// Mitsubishi GX Works2 project: KME Straw Machine   PLC: FX3U/FX3UC

PROGRAM MAIN
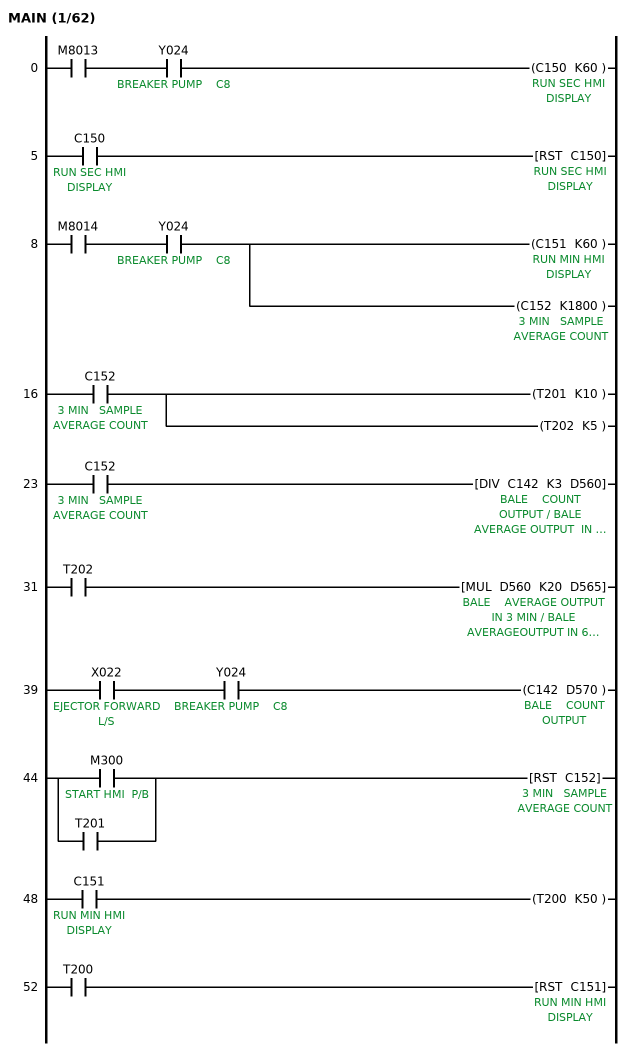
0     LD      M8013
      AND     Y024  ; BREAKER PUMP    C8
      OUT     C150 K60  ; RUN SEC HMI     DISPLAY
5     LD      C150  ; RUN SEC HMI     DISPLAY
      RST     C150  ; RUN SEC HMI     DISPLAY
8     LD      M8014
      AND     Y024  ; BREAKER PUMP    C8
      OUT     C151 K60  ; RUN MIN HMI     DISPLAY
      OUT     C152 K1800  ; 3 MIN   SAMPLE  AVERAGE COUNT
16    LD      C152  ; 3 MIN   SAMPLE  AVERAGE COUNT
      OUT     T201 K10
      OUT     T202 K5
23    LD      C152  ; 3 MIN   SAMPLE  AVERAGE COUNT
      DIV     C142 K3 D560  ; BALE    COUNT   OUTPUT / BALE    AVERAGE OUTPUT  IN 3 MIN
31    LD      T202
      MUL     D560 K20 D565  ; BALE     AVERAGEOUTPUT IN 60 MIN
39    LD      X022  ; EJECTOR FORWARD L/S
      AND     Y024  ; BREAKER PUMP    C8
      OUT     C142 D570  ; BALE    COUNT   OUTPUT
44    LD      M300  ; START HMI  P/B
      OR      T201
      RST     C152  ; 3 MIN   SAMPLE  AVERAGE COUNT
48    LD      C151  ; RUN MIN HMI     DISPLAY
      OUT     T200 K50
52    LD      T200
      RST     C151  ; RUN MIN HMI     DISPLAY
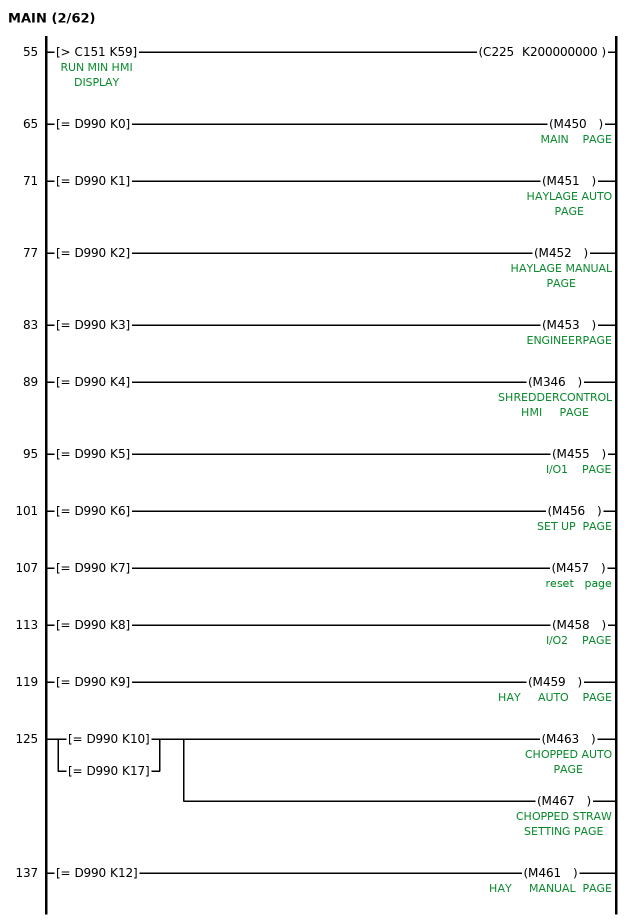
55    LD>     C151 K59  ; RUN MIN HMI     DISPLAY
      OUT     C225 K200000000
65    LD=     D990 K0
      OUT     M450  ; MAIN    PAGE
71    LD=     D990 K1
      OUT     M451  ; HAYLAGE AUTO    PAGE
77    LD=     D990 K2
      OUT     M452  ; HAYLAGE MANUAL  PAGE
83    LD=     D990 K3
      OUT     M453  ; ENGINEERPAGE
89    LD=     D990 K4
      OUT     M346  ; SHREDDERCONTROL HMI     PAGE
95    LD=     D990 K5
      OUT     M455  ; I/O1    PAGE
101   LD=     D990 K6
      OUT     M456  ; SET UP  PAGE
107   LD=     D990 K7
      OUT     M457  ; reset   page
113   LD=     D990 K8
      OUT     M458  ; I/O2    PAGE
119   LD=     D990 K9
      OUT     M459  ; HAY     AUTO    PAGE
125   LD=     D990 K10
      OR=     D990 K17
      OUT     M463  ; CHOPPED AUTO    PAGE
      OUT     M467  ; CHOPPED STRAW   SETTING PAGE
137   LD=     D990 K12
      OUT     M461  ; HAY     MANUAL  PAGE
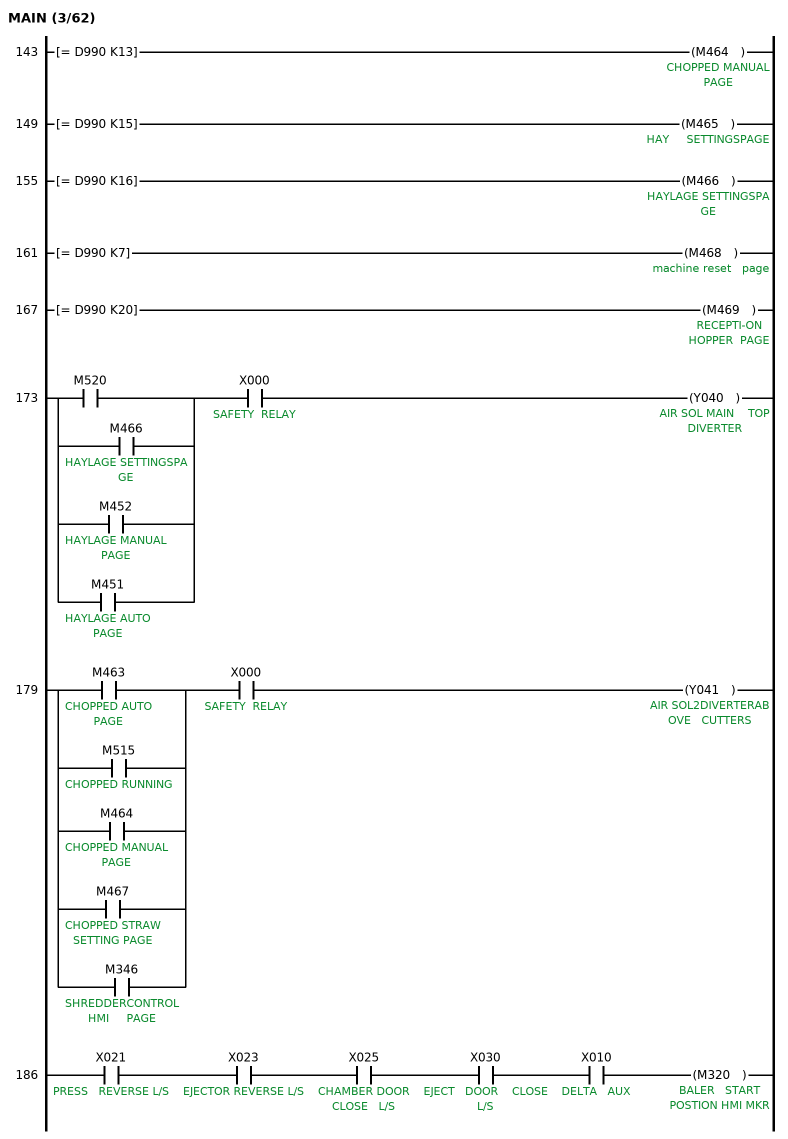
143   LD=     D990 K13
      OUT     M464  ; CHOPPED MANUAL  PAGE
149   LD=     D990 K15
      OUT     M465  ; HAY     SETTINGSPAGE
155   LD=     D990 K16
      OUT     M466  ; HAYLAGE SETTINGSPAGE
161   LD=     D990 K7
      OUT     M468  ; machine reset   page
167   LD=     D990 K20
      OUT     M469  ; RECEPTI-ON      HOPPER  PAGE
173   LD      M520
      OR      M466  ; HAYLAGE SETTINGSPAGE
      OR      M452  ; HAYLAGE MANUAL  PAGE
      OR      M451  ; HAYLAGE AUTO    PAGE
      AND     X000  ; SAFETY  RELAY
      OUT     Y040  ; AIR SOL MAIN    TOP     DIVERTER
179   LD      M463  ; CHOPPED AUTO    PAGE
      OR      M515  ; CHOPPED RUNNING
      OR      M464  ; CHOPPED MANUAL  PAGE
      OR      M467  ; CHOPPED STRAW   SETTING PAGE
      OR      M346  ; SHREDDERCONTROL HMI     PAGE
      AND     X000  ; SAFETY  RELAY
      OUT     Y041  ; AIR SOL2DIVERTERABOVE   CUTTERS
186   LD      X021  ; PRESS   REVERSE L/S
      AND     X023  ; EJECTOR REVERSE L/S
      AND     X025  ; CHAMBER DOOR    CLOSE   L/S
      AND     X030  ; EJECT   DOOR    CLOSE L/S
      AND     X010  ; DELTA   AUX
      OUT     M320  ; BALER   START   POSTION HMI MKR
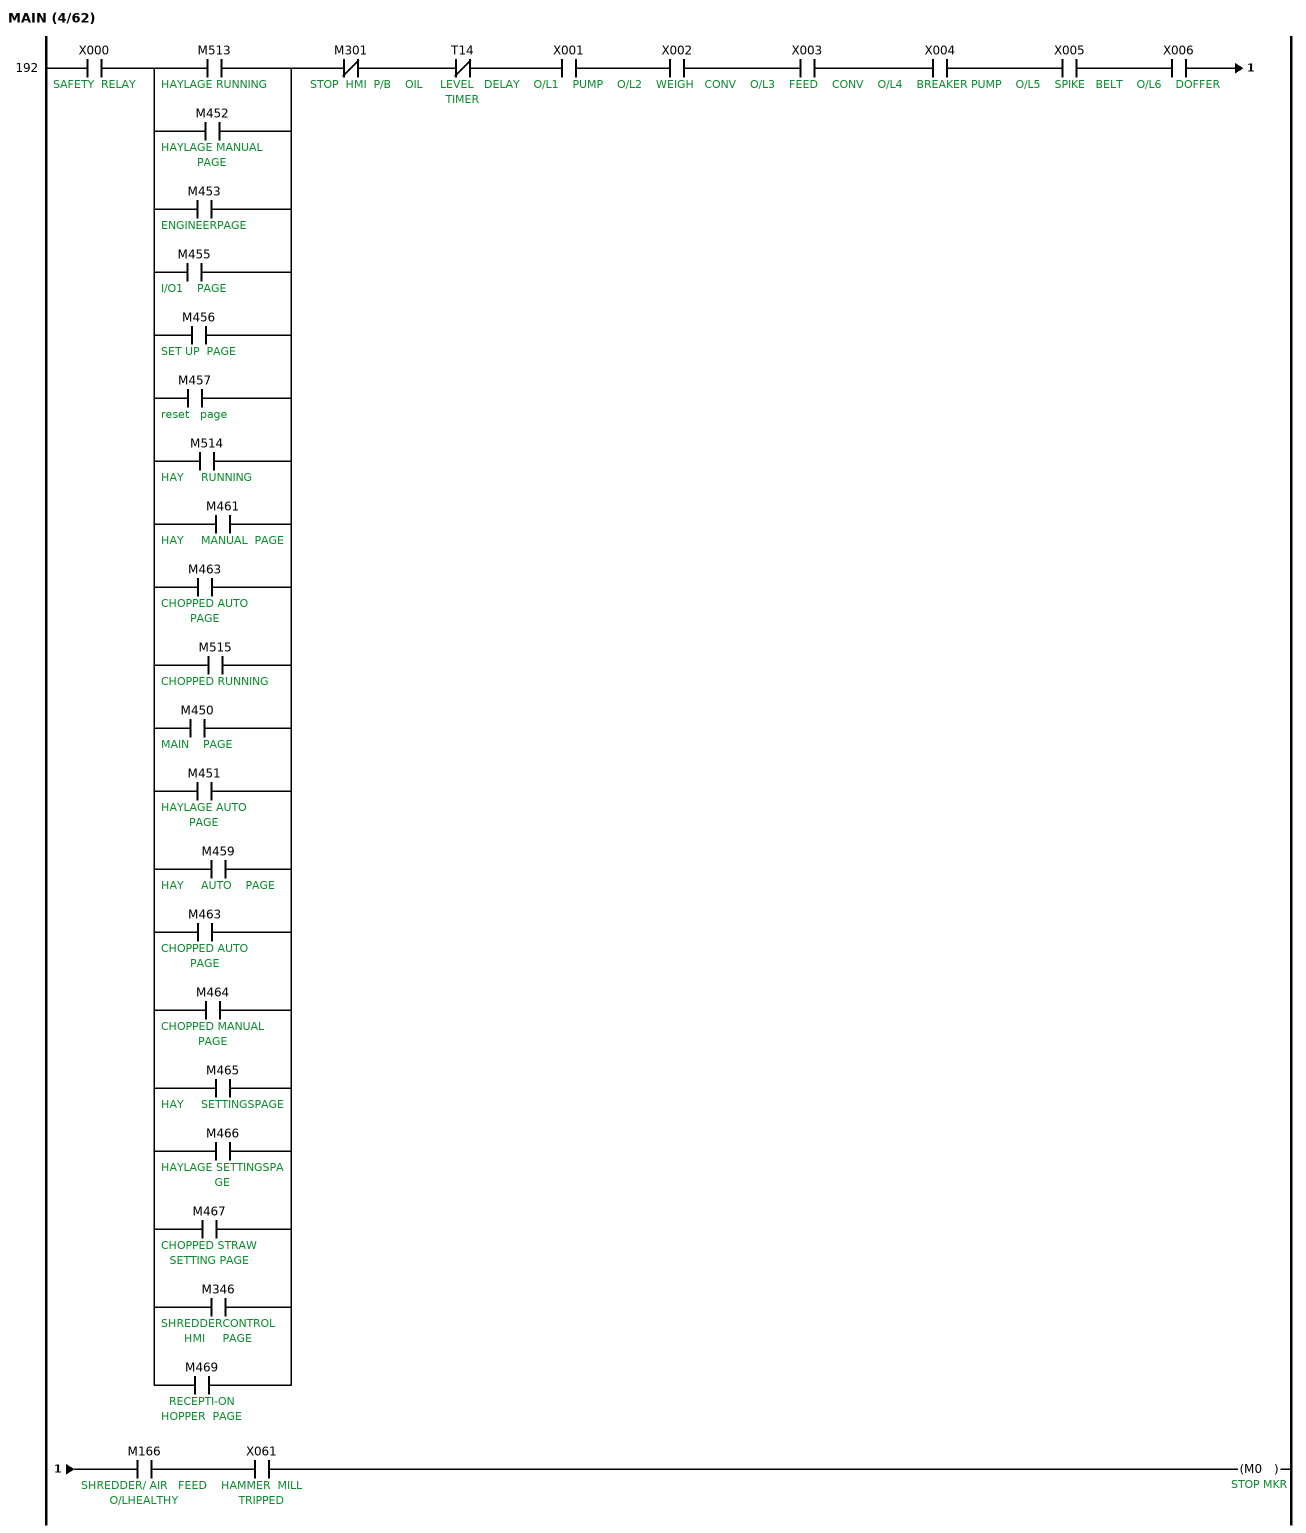
192   LD      X000  ; SAFETY  RELAY
      LD      M513  ; HAYLAGE RUNNING
      OR      M452  ; HAYLAGE MANUAL  PAGE
      OR      M453  ; ENGINEERPAGE
      OR      M455  ; I/O1    PAGE
      OR      M456  ; SET UP  PAGE
      OR      M457  ; reset   page
      OR      M514  ; HAY     RUNNING
      OR      M461  ; HAY     MANUAL  PAGE
      OR      M463  ; CHOPPED AUTO    PAGE
      OR      M515  ; CHOPPED RUNNING
      OR      M450  ; MAIN    PAGE
      OR      M451  ; HAYLAGE AUTO    PAGE
      OR      M459  ; HAY     AUTO    PAGE
      OR      M463  ; CHOPPED AUTO    PAGE
      OR      M464  ; CHOPPED MANUAL  PAGE
      OR      M465  ; HAY     SETTINGSPAGE
      OR      M466  ; HAYLAGE SETTINGSPAGE
      OR      M467  ; CHOPPED STRAW   SETTING PAGE
      OR      M346  ; SHREDDERCONTROL HMI     PAGE
      OR      M469  ; RECEPTI-ON      HOPPER  PAGE
      ANB
      ANI     M301  ; STOP  HMI  P/B
      ANI     T14  ; OIL     LEVEL   DELAY   TIMER
      AND     X001  ; O/L1    PUMP
      AND     X002  ; O/L2    WEIGH   CONV
      AND     X003  ; O/L3    FEED    CONV
      AND     X004  ; O/L4    BREAKER PUMP
      AND     X005  ; O/L5    SPIKE   BELT
      AND     X006  ; O/L6    DOFFER
      AND     M166  ; SHREDDER/ AIR   FEED O/LHEALTHY
      AND     X061  ; HAMMER  MILL    TRIPPED
      OUT     M0  ; STOP MKR
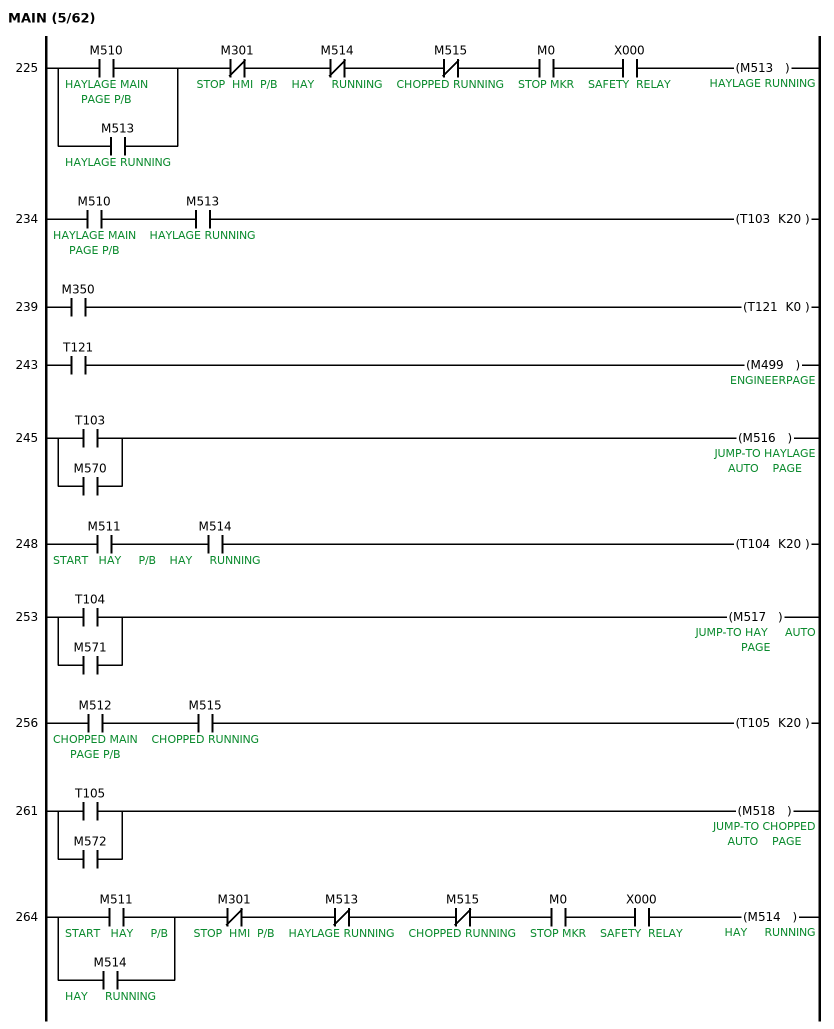
225   LD      M510  ; HAYLAGE MAIN    PAGE P/B
      OR      M513  ; HAYLAGE RUNNING
      ANI     M301  ; STOP  HMI  P/B
      ANI     M514  ; HAY     RUNNING
      ANI     M515  ; CHOPPED RUNNING
      AND     M0  ; STOP MKR
      AND     X000  ; SAFETY  RELAY
      OUT     M513  ; HAYLAGE RUNNING
234   LD      M510  ; HAYLAGE MAIN    PAGE P/B
      AND     M513  ; HAYLAGE RUNNING
      OUT     T103 K20
239   LD      M350
      OUT     T121 K0
243   LD      T121
      OUT     M499  ; ENGINEERPAGE
245   LD      T103
      OR      M570
      OUT     M516  ; JUMP-TO HAYLAGE AUTO    PAGE
248   LD      M511  ; START   HAY     P/B
      AND     M514  ; HAY     RUNNING
      OUT     T104 K20
253   LD      T104
      OR      M571
      OUT     M517  ; JUMP-TO HAY     AUTO    PAGE
256   LD      M512  ; CHOPPED MAIN    PAGE P/B
      AND     M515  ; CHOPPED RUNNING
      OUT     T105 K20
261   LD      T105
      OR      M572
      OUT     M518  ; JUMP-TO CHOPPED AUTO    PAGE
264   LD      M511  ; START   HAY     P/B
      OR      M514  ; HAY     RUNNING
      ANI     M301  ; STOP  HMI  P/B
      ANI     M513  ; HAYLAGE RUNNING
      ANI     M515  ; CHOPPED RUNNING
      AND     M0  ; STOP MKR
      AND     X000  ; SAFETY  RELAY
      OUT     M514  ; HAY     RUNNING
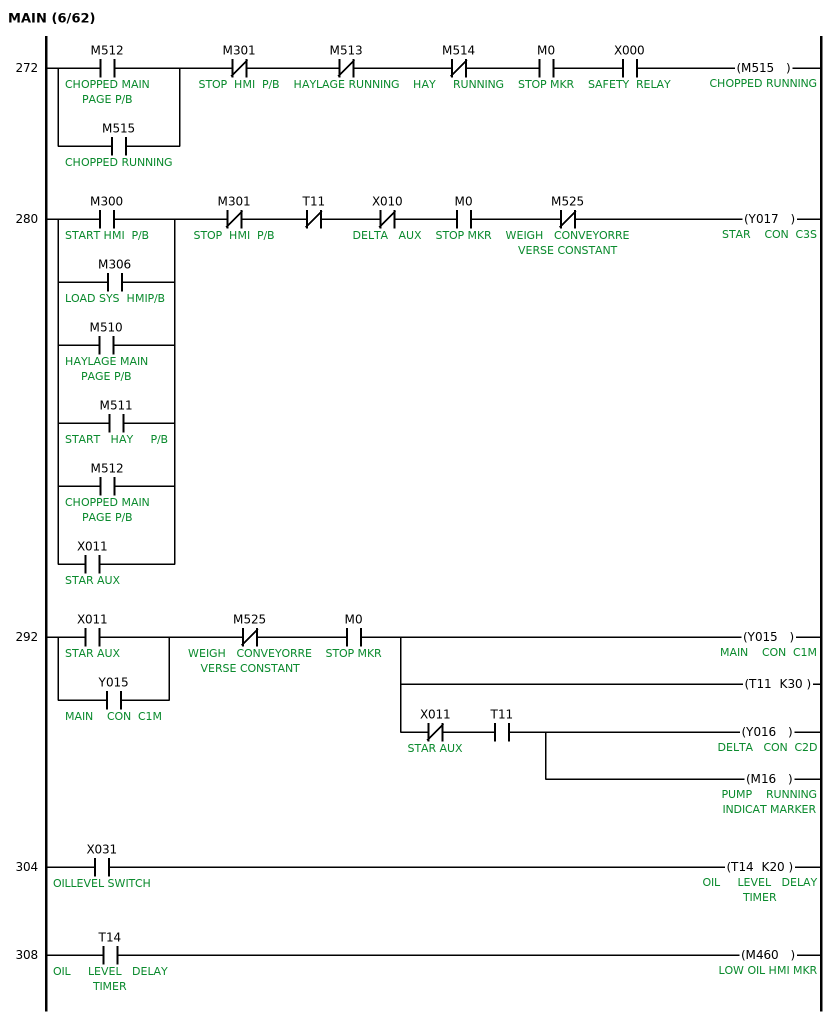
272   LD      M512  ; CHOPPED MAIN    PAGE P/B
      OR      M515  ; CHOPPED RUNNING
      ANI     M301  ; STOP  HMI  P/B
      ANI     M513  ; HAYLAGE RUNNING
      ANI     M514  ; HAY     RUNNING
      AND     M0  ; STOP MKR
      AND     X000  ; SAFETY  RELAY
      OUT     M515  ; CHOPPED RUNNING
280   LD      M300  ; START HMI  P/B
      OR      M306  ; LOAD SYS  HMIP/B
      OR      M510  ; HAYLAGE MAIN    PAGE P/B
      OR      M511  ; START   HAY     P/B
      OR      M512  ; CHOPPED MAIN    PAGE P/B
      OR      X011  ; STAR AUX
      ANI     M301  ; STOP  HMI  P/B
      ANI     T11
      ANI     X010  ; DELTA   AUX
      AND     M0  ; STOP MKR
      ANI     M525  ; WEIGH   CONVEYORREVERSE CONSTANT
      OUT     Y017  ; STAR    CON  C3S
292   LD      X011  ; STAR AUX
      OR      Y015  ; MAIN    CON  C1M
      ANI     M525  ; WEIGH   CONVEYORREVERSE CONSTANT
      AND     M0  ; STOP MKR
      OUT     Y015  ; MAIN    CON  C1M
      OUT     T11 K30
      ANI     X011  ; STAR AUX
      AND     T11
      OUT     Y016  ; DELTA   CON  C2D
      OUT     M16  ; PUMP    RUNNING INDICAT MARKER
304   LD      X031  ; OILLEVEL SWITCH
      OUT     T14 K20  ; OIL     LEVEL   DELAY   TIMER
308   LD      T14  ; OIL     LEVEL   DELAY   TIMER
      OUT     M460  ; LOW OIL HMI MKR
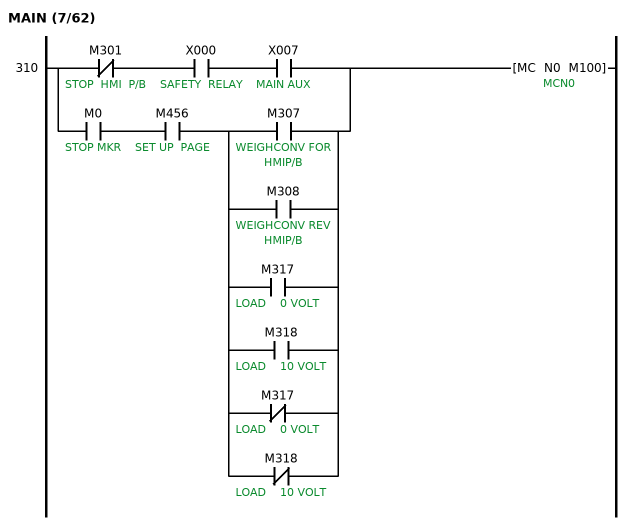
310   LDI     M301  ; STOP  HMI  P/B
      AND     X000  ; SAFETY  RELAY
      AND     X007  ; MAIN AUX
      LD      M0  ; STOP MKR
      AND     M456  ; SET UP  PAGE
      LD      M307  ; WEIGHCONV FOR   HMIP/B
      OR      M308  ; WEIGHCONV REV   HMIP/B
      OR      M317  ; LOAD    0 VOLT
      OR      M318  ; LOAD    10 VOLT
      ORI     M317  ; LOAD    0 VOLT
      ORI     M318  ; LOAD    10 VOLT
      ANB
      ORB
      MC      N0 M100  ; MCN0
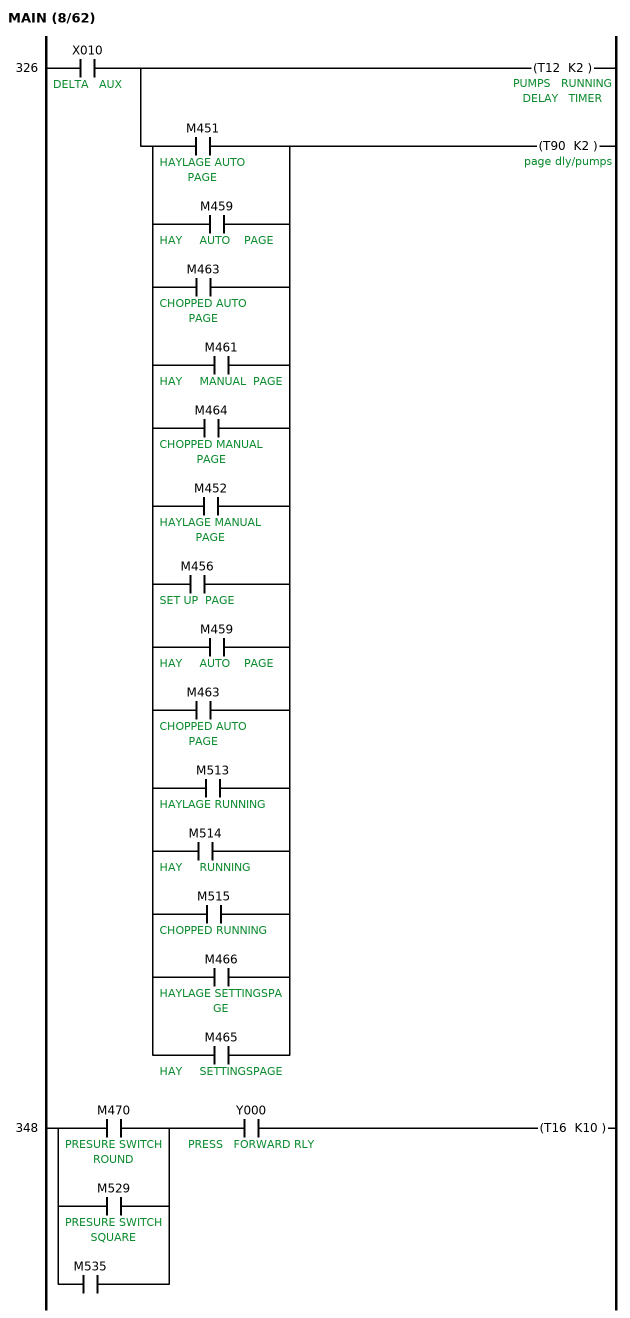
326   LD      X010  ; DELTA   AUX
      OUT     T12 K2  ; PUMPS   RUNNING DELAY   TIMER
      LD      M451  ; HAYLAGE AUTO    PAGE
      OR      M459  ; HAY     AUTO    PAGE
      OR      M463  ; CHOPPED AUTO    PAGE
      OR      M461  ; HAY     MANUAL  PAGE
      OR      M464  ; CHOPPED MANUAL  PAGE
      OR      M452  ; HAYLAGE MANUAL  PAGE
      OR      M456  ; SET UP  PAGE
      OR      M459  ; HAY     AUTO    PAGE
      OR      M463  ; CHOPPED AUTO    PAGE
      OR      M513  ; HAYLAGE RUNNING
      OR      M514  ; HAY     RUNNING
      OR      M515  ; CHOPPED RUNNING
      OR      M466  ; HAYLAGE SETTINGSPAGE
      OR      M465  ; HAY     SETTINGSPAGE
      ANB
      OUT     T90 K2  ; page dly/pumps
348   LD      M470  ; PRESURE SWITCH  ROUND
      OR      M529  ; PRESURE SWITCH  SQUARE
      OR      M535
      AND     Y000  ; PRESS   FORWARD RLY
      OUT     T16 K10
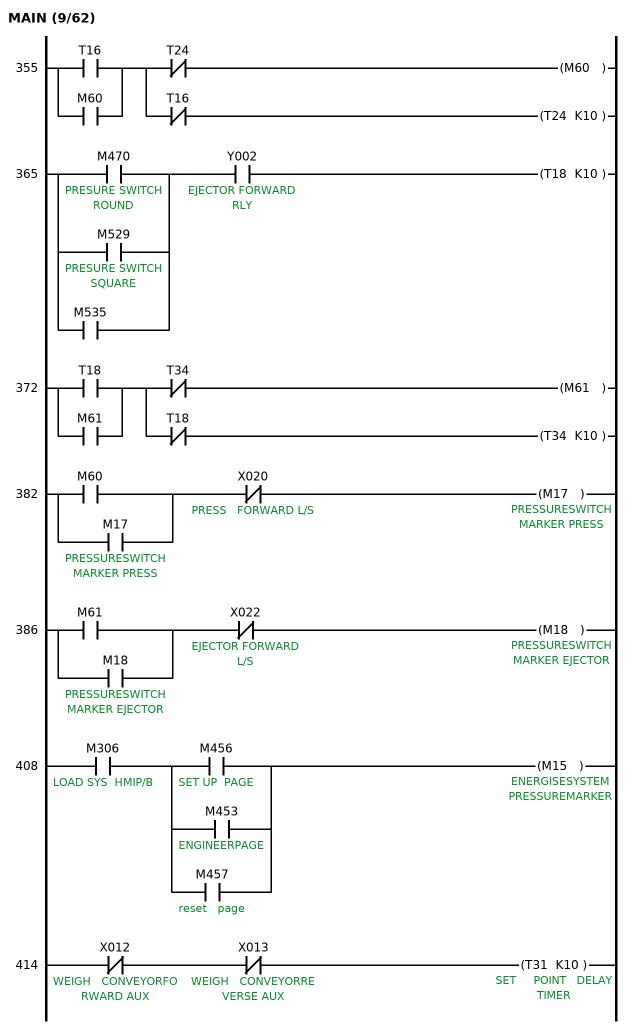
355   LD      T16
      OR      M60
      MPS
      ANI     T24
      OUT     M60
      MPP
      ANI     T16
      OUT     T24 K10
365   LD      M470  ; PRESURE SWITCH  ROUND
      OR      M529  ; PRESURE SWITCH  SQUARE
      OR      M535
      AND     Y002  ; EJECTOR FORWARD RLY
      OUT     T18 K10
372   LD      T18
      OR      M61
      MPS
      ANI     T34
      OUT     M61
      MPP
      ANI     T18
      OUT     T34 K10
382   LD      M60
      OR      M17  ; PRESSURESWITCH  MARKER PRESS
      ANI     X020  ; PRESS   FORWARD L/S
      OUT     M17  ; PRESSURESWITCH  MARKER PRESS
386   LD      M61
      OR      M18  ; PRESSURESWITCH  MARKER EJECTOR
      ANI     X022  ; EJECTOR FORWARD L/S
      OUT     M18  ; PRESSURESWITCH  MARKER EJECTOR
408   LD      M306  ; LOAD SYS  HMIP/B
      LD      M456  ; SET UP  PAGE
      OR      M453  ; ENGINEERPAGE
      OR      M457  ; reset   page
      ANB
      OUT     M15  ; ENERGISESYSTEM  PRESSUREMARKER
414   LDI     X012  ; WEIGH   CONVEYORFORWARD AUX
      ANI     X013  ; WEIGH   CONVEYORREVERSE AUX
      OUT     T31 K10  ; SET     POINT   DELAY   TIMER
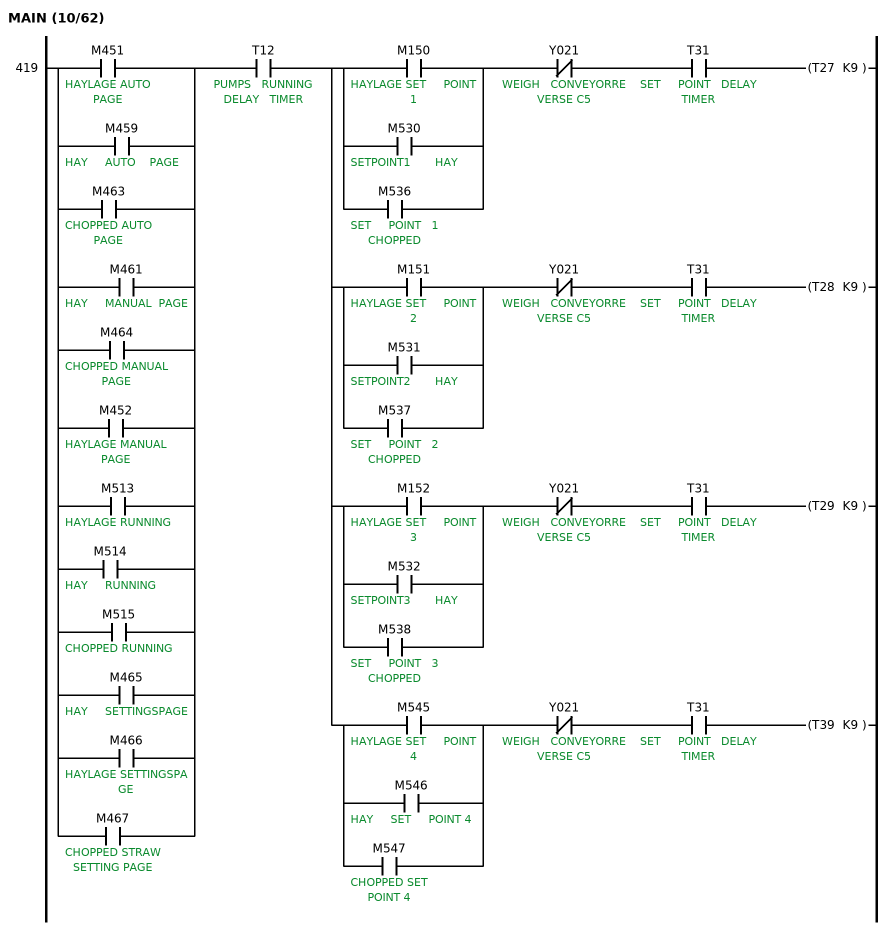
419   LD      M451  ; HAYLAGE AUTO    PAGE
      OR      M459  ; HAY     AUTO    PAGE
      OR      M463  ; CHOPPED AUTO    PAGE
      OR      M461  ; HAY     MANUAL  PAGE
      OR      M464  ; CHOPPED MANUAL  PAGE
      OR      M452  ; HAYLAGE MANUAL  PAGE
      OR      M513  ; HAYLAGE RUNNING
      OR      M514  ; HAY     RUNNING
      OR      M515  ; CHOPPED RUNNING
      OR      M465  ; HAY     SETTINGSPAGE
      OR      M466  ; HAYLAGE SETTINGSPAGE
      OR      M467  ; CHOPPED STRAW   SETTING PAGE
      AND     T12  ; PUMPS   RUNNING DELAY   TIMER
      MPS
      LD      M150  ; HAYLAGE SET     POINT 1
      OR      M530  ; SETPOINT1       HAY
      OR      M536  ; SET     POINT   1       CHOPPED
      ANB
      ANI     Y021  ; WEIGH   CONVEYORREVERSE C5
      AND     T31  ; SET     POINT   DELAY   TIMER
      OUT     T27 K9
      MRD
      LD      M151  ; HAYLAGE SET     POINT 2
      OR      M531  ; SETPOINT2       HAY
      OR      M537  ; SET     POINT   2       CHOPPED
      ANB
      ANI     Y021  ; WEIGH   CONVEYORREVERSE C5
      AND     T31  ; SET     POINT   DELAY   TIMER
      OUT     T28 K9
      MRD
      LD      M152  ; HAYLAGE SET     POINT 3
      OR      M532  ; SETPOINT3       HAY
      OR      M538  ; SET     POINT   3       CHOPPED
      ANB
      ANI     Y021  ; WEIGH   CONVEYORREVERSE C5
      AND     T31  ; SET     POINT   DELAY   TIMER
      OUT     T29 K9
      MPP
      LD      M545  ; HAYLAGE SET     POINT 4
      OR      M546  ; HAY     SET     POINT 4
      OR      M547  ; CHOPPED SET     POINT 4
      ANB
      ANI     Y021  ; WEIGH   CONVEYORREVERSE C5
      AND     T31  ; SET     POINT   DELAY   TIMER
      OUT     T39 K9
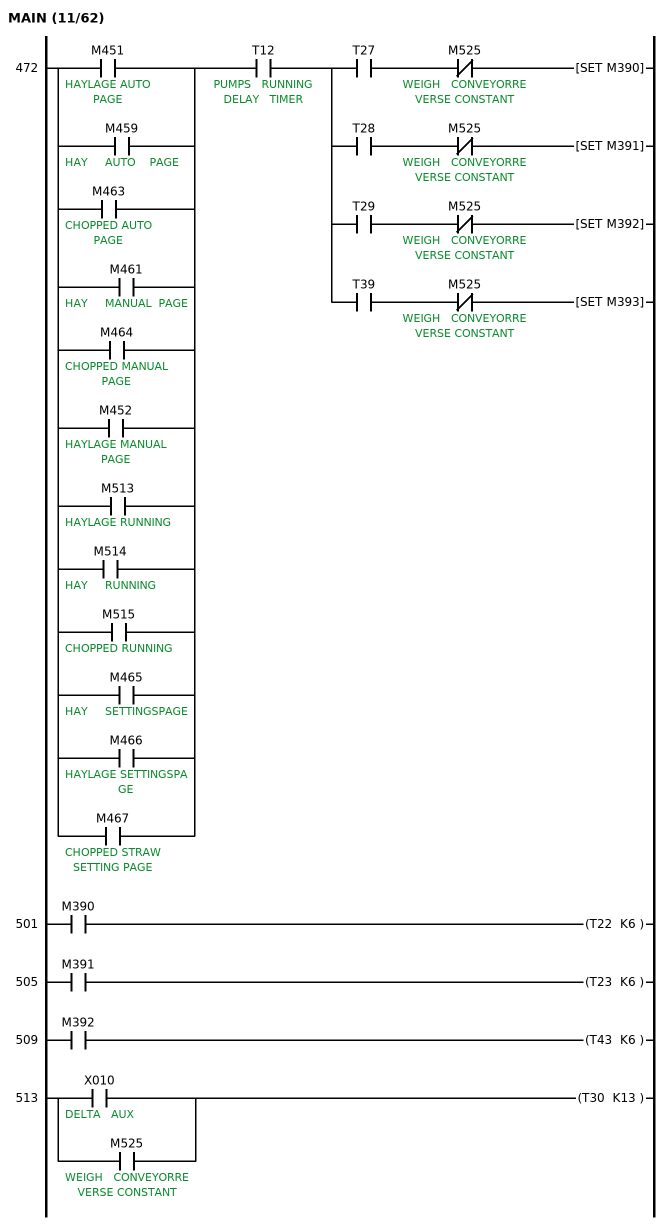
472   LD      M451  ; HAYLAGE AUTO    PAGE
      OR      M459  ; HAY     AUTO    PAGE
      OR      M463  ; CHOPPED AUTO    PAGE
      OR      M461  ; HAY     MANUAL  PAGE
      OR      M464  ; CHOPPED MANUAL  PAGE
      OR      M452  ; HAYLAGE MANUAL  PAGE
      OR      M513  ; HAYLAGE RUNNING
      OR      M514  ; HAY     RUNNING
      OR      M515  ; CHOPPED RUNNING
      OR      M465  ; HAY     SETTINGSPAGE
      OR      M466  ; HAYLAGE SETTINGSPAGE
      OR      M467  ; CHOPPED STRAW   SETTING PAGE
      AND     T12  ; PUMPS   RUNNING DELAY   TIMER
      MPS
      AND     T27
      ANI     M525  ; WEIGH   CONVEYORREVERSE CONSTANT
      SET     M390
      MRD
      AND     T28
      ANI     M525  ; WEIGH   CONVEYORREVERSE CONSTANT
      SET     M391
      MRD
      AND     T29
      ANI     M525  ; WEIGH   CONVEYORREVERSE CONSTANT
      SET     M392
      MPP
      AND     T39
      ANI     M525  ; WEIGH   CONVEYORREVERSE CONSTANT
      SET     M393
501   LD      M390
      OUT     T22 K6
505   LD      M391
      OUT     T23 K6
509   LD      M392
      OUT     T43 K6
513   LD      X010  ; DELTA   AUX
      OR      M525  ; WEIGH   CONVEYORREVERSE CONSTANT
      OUT     T30 K13
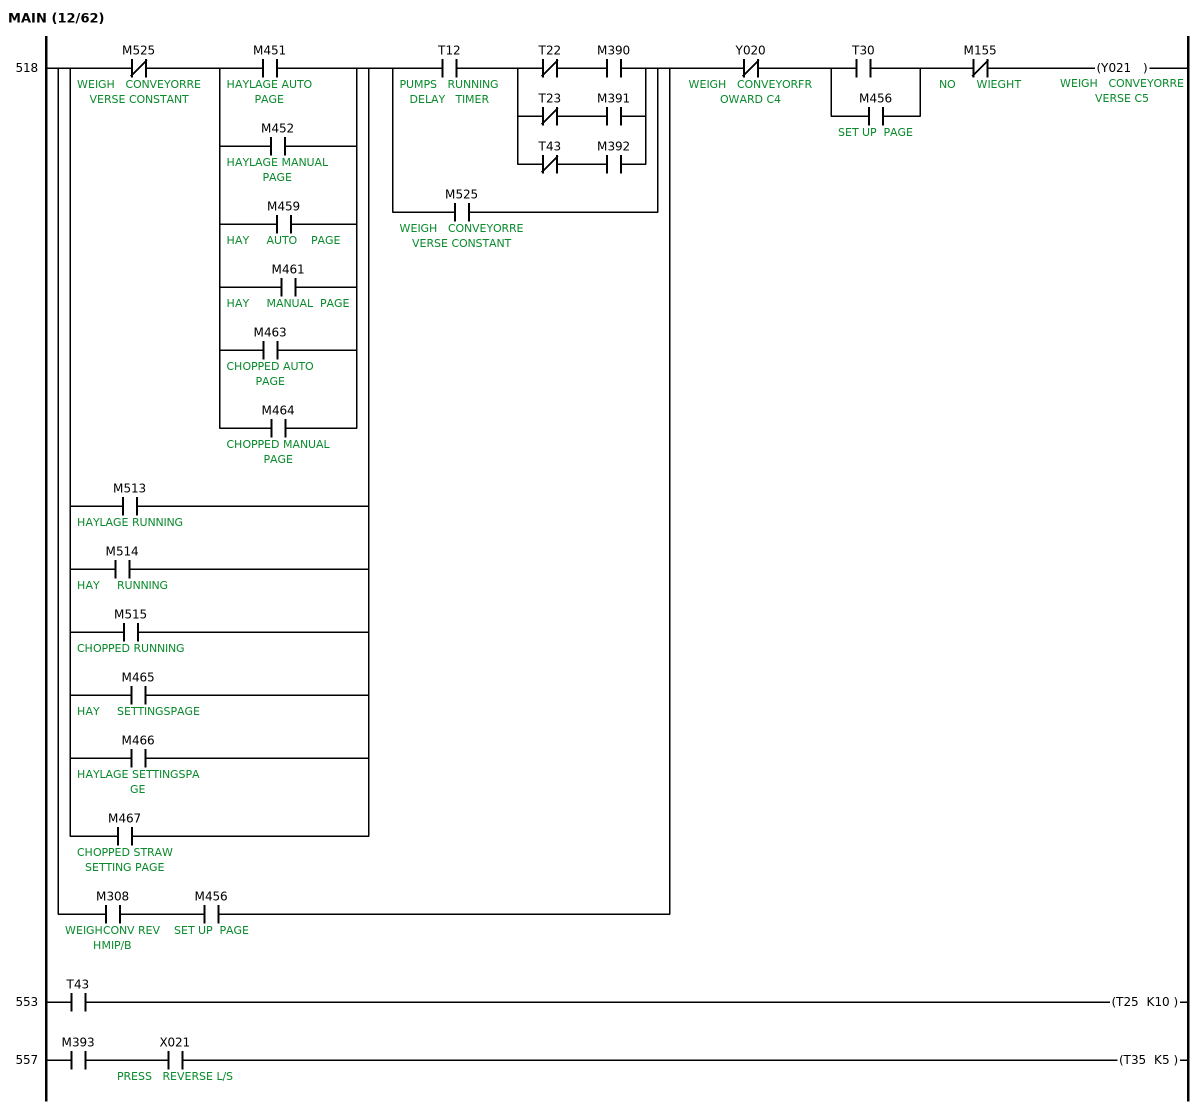
518   LDI     M525  ; WEIGH   CONVEYORREVERSE CONSTANT
      LD      M451  ; HAYLAGE AUTO    PAGE
      OR      M452  ; HAYLAGE MANUAL  PAGE
      OR      M459  ; HAY     AUTO    PAGE
      OR      M461  ; HAY     MANUAL  PAGE
      OR      M463  ; CHOPPED AUTO    PAGE
      OR      M464  ; CHOPPED MANUAL  PAGE
      ANB
      OR      M513  ; HAYLAGE RUNNING
      OR      M514  ; HAY     RUNNING
      OR      M515  ; CHOPPED RUNNING
      OR      M465  ; HAY     SETTINGSPAGE
      OR      M466  ; HAYLAGE SETTINGSPAGE
      OR      M467  ; CHOPPED STRAW   SETTING PAGE
      LD      T12  ; PUMPS   RUNNING DELAY   TIMER
      LDI     T22
      AND     M390
      LDI     T23
      AND     M391
      ORB
      LDI     T43
      AND     M392
      ORB
      ANB
      OR      M525  ; WEIGH   CONVEYORREVERSE CONSTANT
      ANB
      LD      M308  ; WEIGHCONV REV   HMIP/B
      AND     M456  ; SET UP  PAGE
      ORB
      ANI     Y020  ; WEIGH   CONVEYORFROWARD C4
      LD      T30
      OR      M456  ; SET UP  PAGE
      ANB
      ANI     M155  ; NO      WIEGHT
      OUT     Y021  ; WEIGH   CONVEYORREVERSE C5
553   LD      T43
      OUT     T25 K10
557   LD      M393
      AND     X021  ; PRESS   REVERSE L/S
      OUT     T35 K5
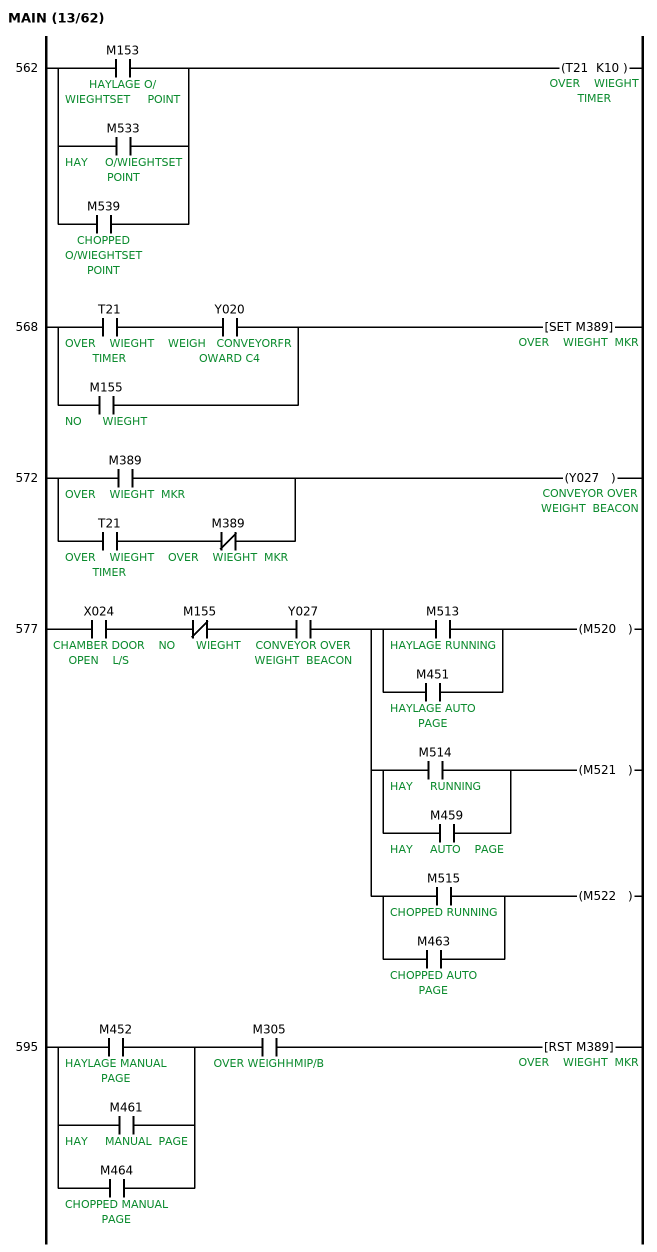
562   LD      M153  ; HAYLAGE O/WIEGHTSET     POINT
      OR      M533  ; HAY     O/WIEGHTSET     POINT
      OR      M539  ; CHOPPED O/WIEGHTSET     POINT
      OUT     T21 K10  ; OVER    WIEGHT  TIMER
568   LD      T21  ; OVER    WIEGHT  TIMER
      AND     Y020  ; WEIGH   CONVEYORFROWARD C4
      OR      M155  ; NO      WIEGHT
      SET     M389  ; OVER    WIEGHT  MKR
572   LD      M389  ; OVER    WIEGHT  MKR
      LD      T21  ; OVER    WIEGHT  TIMER
      ANI     M389  ; OVER    WIEGHT  MKR
      ORB
      OUT     Y027  ; CONVEYOR OVER   WEIGHT  BEACON
577   LD      X024  ; CHAMBER DOOR    OPEN    L/S
      ANI     M155  ; NO      WIEGHT
      AND     Y027  ; CONVEYOR OVER   WEIGHT  BEACON
      MPS
      LD      M513  ; HAYLAGE RUNNING
      OR      M451  ; HAYLAGE AUTO    PAGE
      ANB
      OUT     M520
      MRD
      LD      M514  ; HAY     RUNNING
      OR      M459  ; HAY     AUTO    PAGE
      ANB
      OUT     M521
      MPP
      LD      M515  ; CHOPPED RUNNING
      OR      M463  ; CHOPPED AUTO    PAGE
      ANB
      OUT     M522
595   LD      M452  ; HAYLAGE MANUAL  PAGE
      OR      M461  ; HAY     MANUAL  PAGE
      OR      M464  ; CHOPPED MANUAL  PAGE
      AND     M305  ; OVER WEIGHHMIP/B
      RST     M389  ; OVER    WIEGHT  MKR
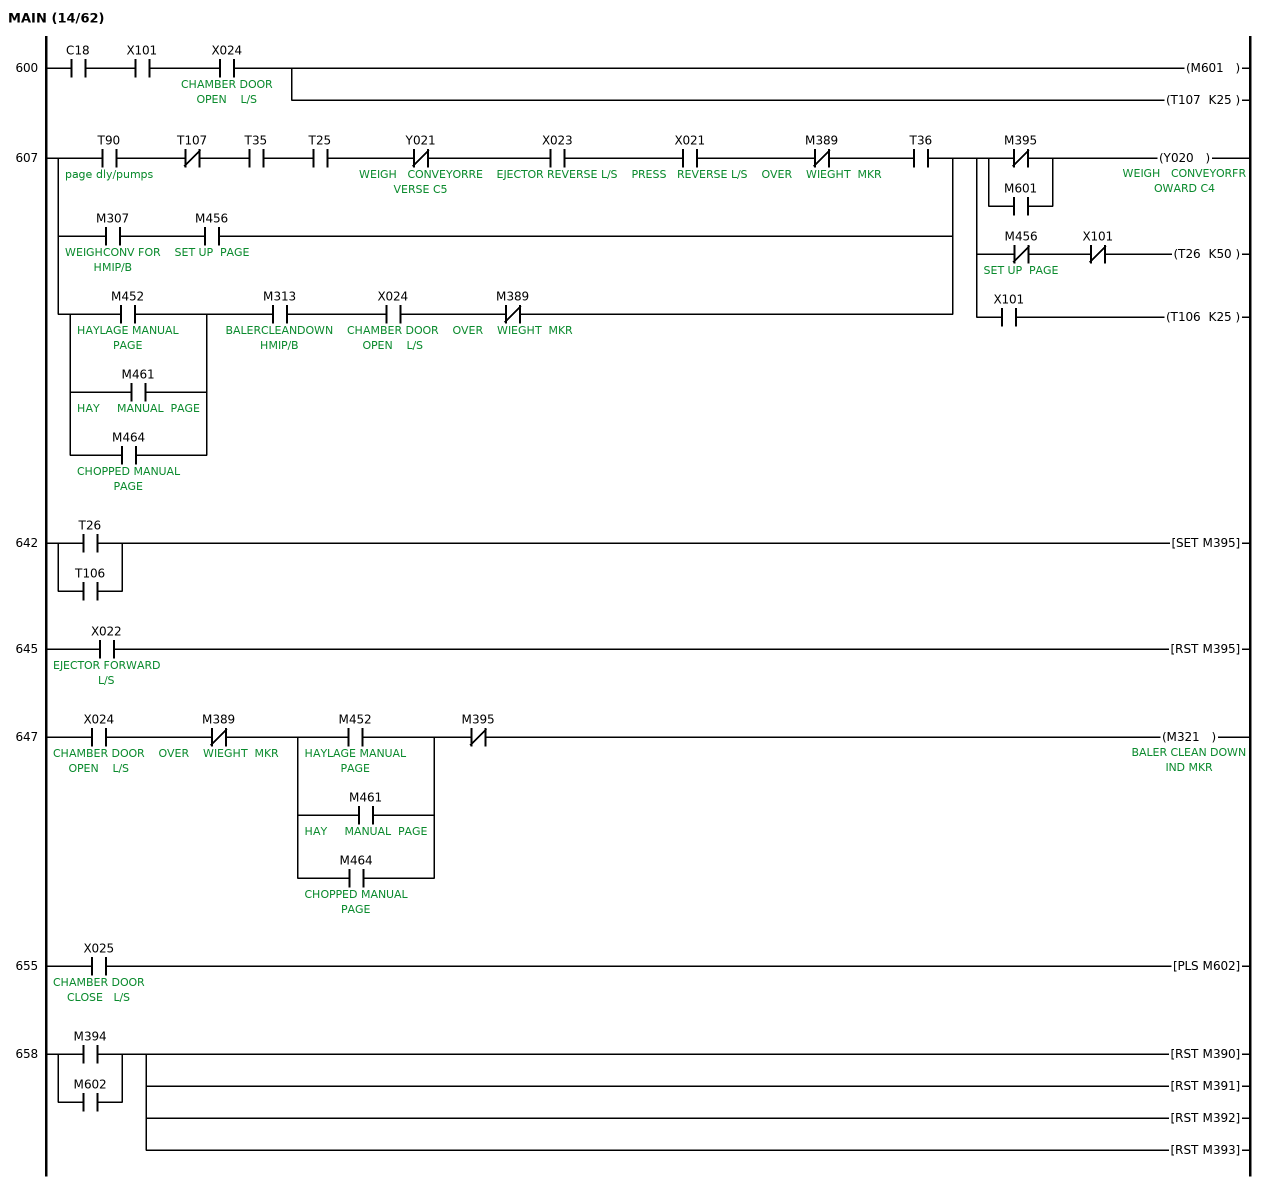
600   LD      C18
      AND     X101
      AND     X024  ; CHAMBER DOOR    OPEN    L/S
      OUT     M601
      OUT     T107 K25
607   LD      T90  ; page dly/pumps
      ANI     T107
      AND     T35
      AND     T25
      ANI     Y021  ; WEIGH   CONVEYORREVERSE C5
      AND     X023  ; EJECTOR REVERSE L/S
      AND     X021  ; PRESS   REVERSE L/S
      ANI     M389  ; OVER    WIEGHT  MKR
      AND     T36
      LD      M307  ; WEIGHCONV FOR   HMIP/B
      AND     M456  ; SET UP  PAGE
      ORB
      LD      M452  ; HAYLAGE MANUAL  PAGE
      OR      M461  ; HAY     MANUAL  PAGE
      OR      M464  ; CHOPPED MANUAL  PAGE
      AND     M313  ; BALERCLEANDOWN  HMIP/B
      AND     X024  ; CHAMBER DOOR    OPEN    L/S
      ANI     M389  ; OVER    WIEGHT  MKR
      ORB
      MPS
      LDI     M395
      OR      M601
      ANB
      OUT     Y020  ; WEIGH   CONVEYORFROWARD C4
      MRD
      ANI     M456  ; SET UP  PAGE
      ANI     X101
      OUT     T26 K50
      MPP
      AND     X101
      OUT     T106 K25
642   LD      T26
      OR      T106
      SET     M395
645   LD      X022  ; EJECTOR FORWARD L/S
      RST     M395
647   LD      X024  ; CHAMBER DOOR    OPEN    L/S
      ANI     M389  ; OVER    WIEGHT  MKR
      LD      M452  ; HAYLAGE MANUAL  PAGE
      OR      M461  ; HAY     MANUAL  PAGE
      OR      M464  ; CHOPPED MANUAL  PAGE
      ANB
      ANI     M395
      OUT     M321  ; BALER CLEAN DOWN IND MKR
655   LD      X025  ; CHAMBER DOOR    CLOSE   L/S
      PLS     M602
658   LD      M394
      OR      M602
      RST     M390
      RST     M391
      RST     M392
      RST     M393
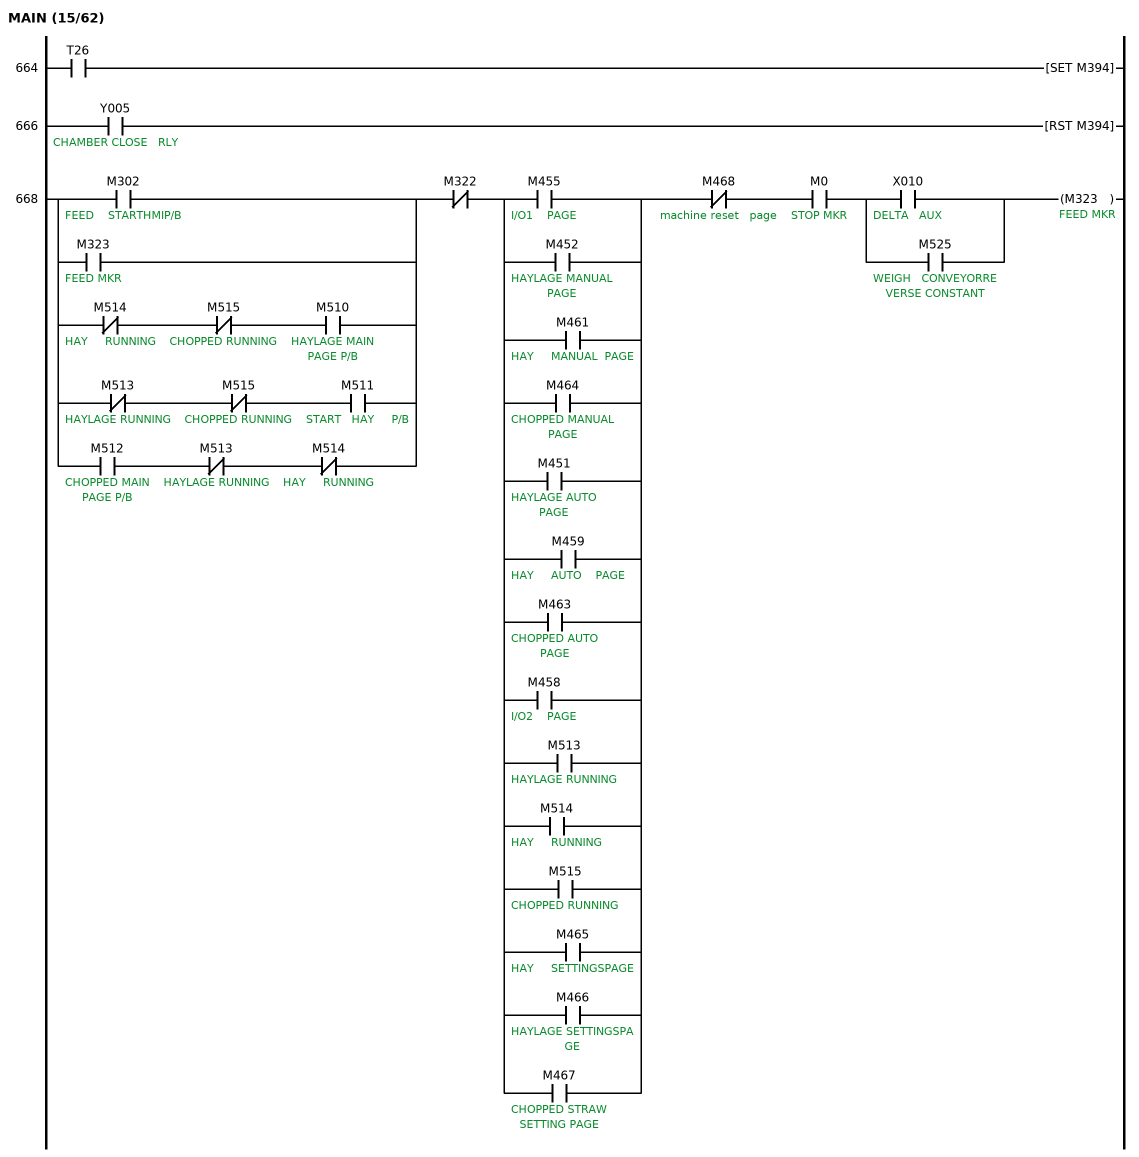
664   LD      T26
      SET     M394
666   LD      Y005  ; CHAMBER CLOSE   RLY
      RST     M394
668   LD      M302  ; FEED    STARTHMIP/B
      OR      M323  ; FEED MKR
      LDI     M514  ; HAY     RUNNING
      ANI     M515  ; CHOPPED RUNNING
      AND     M510  ; HAYLAGE MAIN    PAGE P/B
      ORB
      LDI     M513  ; HAYLAGE RUNNING
      ANI     M515  ; CHOPPED RUNNING
      AND     M511  ; START   HAY     P/B
      ORB
      LD      M512  ; CHOPPED MAIN    PAGE P/B
      ANI     M513  ; HAYLAGE RUNNING
      ANI     M514  ; HAY     RUNNING
      ORB
      ANI     M322
      LD      M455  ; I/O1    PAGE
      OR      M452  ; HAYLAGE MANUAL  PAGE
      OR      M461  ; HAY     MANUAL  PAGE
      OR      M464  ; CHOPPED MANUAL  PAGE
      OR      M451  ; HAYLAGE AUTO    PAGE
      OR      M459  ; HAY     AUTO    PAGE
      OR      M463  ; CHOPPED AUTO    PAGE
      OR      M458  ; I/O2    PAGE
      OR      M513  ; HAYLAGE RUNNING
      OR      M514  ; HAY     RUNNING
      OR      M515  ; CHOPPED RUNNING
      OR      M465  ; HAY     SETTINGSPAGE
      OR      M466  ; HAYLAGE SETTINGSPAGE
      OR      M467  ; CHOPPED STRAW   SETTING PAGE
      ANB
      ANI     M468  ; machine reset   page
      AND     M0  ; STOP MKR
      LD      X010  ; DELTA   AUX
      OR      M525  ; WEIGH   CONVEYORREVERSE CONSTANT
      ANB
      OUT     M323  ; FEED MKR
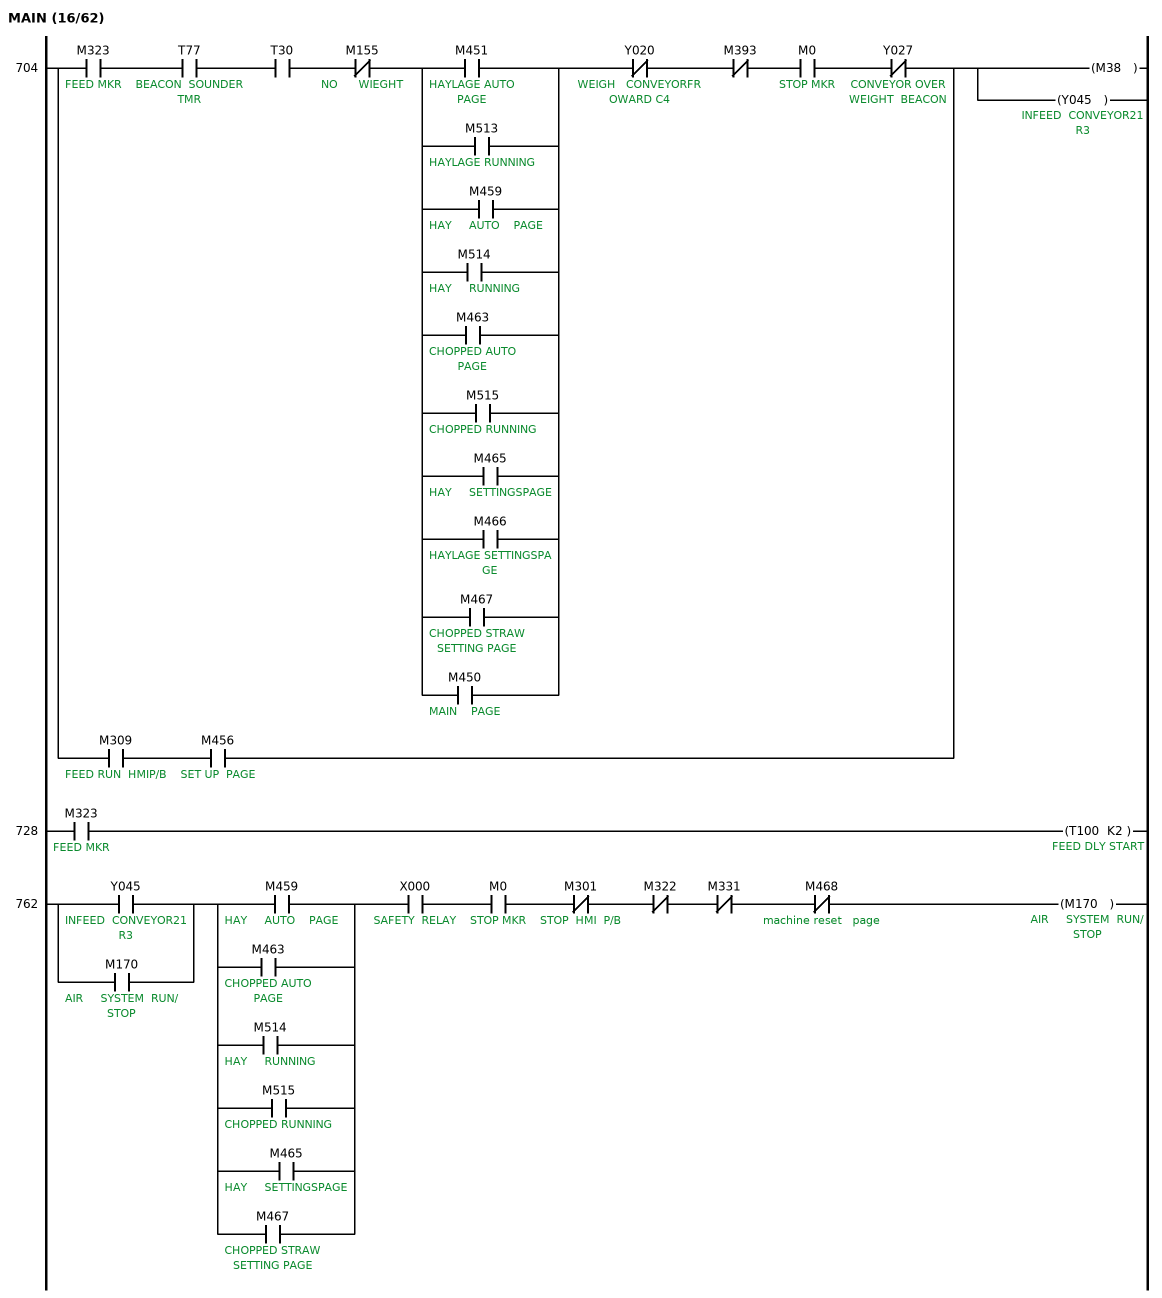
704   LD      M323  ; FEED MKR
      AND     T77  ; BEACON  SOUNDER TMR
      AND     T30
      ANI     M155  ; NO      WIEGHT
      LD      M451  ; HAYLAGE AUTO    PAGE
      OR      M513  ; HAYLAGE RUNNING
      OR      M459  ; HAY     AUTO    PAGE
      OR      M514  ; HAY     RUNNING
      OR      M463  ; CHOPPED AUTO    PAGE
      OR      M515  ; CHOPPED RUNNING
      OR      M465  ; HAY     SETTINGSPAGE
      OR      M466  ; HAYLAGE SETTINGSPAGE
      OR      M467  ; CHOPPED STRAW   SETTING PAGE
      OR      M450  ; MAIN    PAGE
      ANB
      ANI     Y020  ; WEIGH   CONVEYORFROWARD C4
      ANI     M393
      AND     M0  ; STOP MKR
      ANI     Y027  ; CONVEYOR OVER   WEIGHT  BEACON
      LD      M309  ; FEED RUN  HMIP/B
      AND     M456  ; SET UP  PAGE
      ORB
      OUT     M38
      OUT     Y045  ; INFEED  CONVEYOR21R3
728   LD      M323  ; FEED MKR
      OUT     T100 K2  ; FEED DLY START
762   LD      Y045  ; INFEED  CONVEYOR21R3
      OR      M170  ; AIR     SYSTEM  RUN/    STOP
      LD      M459  ; HAY     AUTO    PAGE
      OR      M463  ; CHOPPED AUTO    PAGE
      OR      M514  ; HAY     RUNNING
      OR      M515  ; CHOPPED RUNNING
      OR      M465  ; HAY     SETTINGSPAGE
      OR      M467  ; CHOPPED STRAW   SETTING PAGE
      ANB
      AND     X000  ; SAFETY  RELAY
      AND     M0  ; STOP MKR
      ANI     M301  ; STOP  HMI  P/B
      ANI     M322
      ANI     M331
      ANI     M468  ; machine reset   page
      OUT     M170  ; AIR     SYSTEM  RUN/    STOP
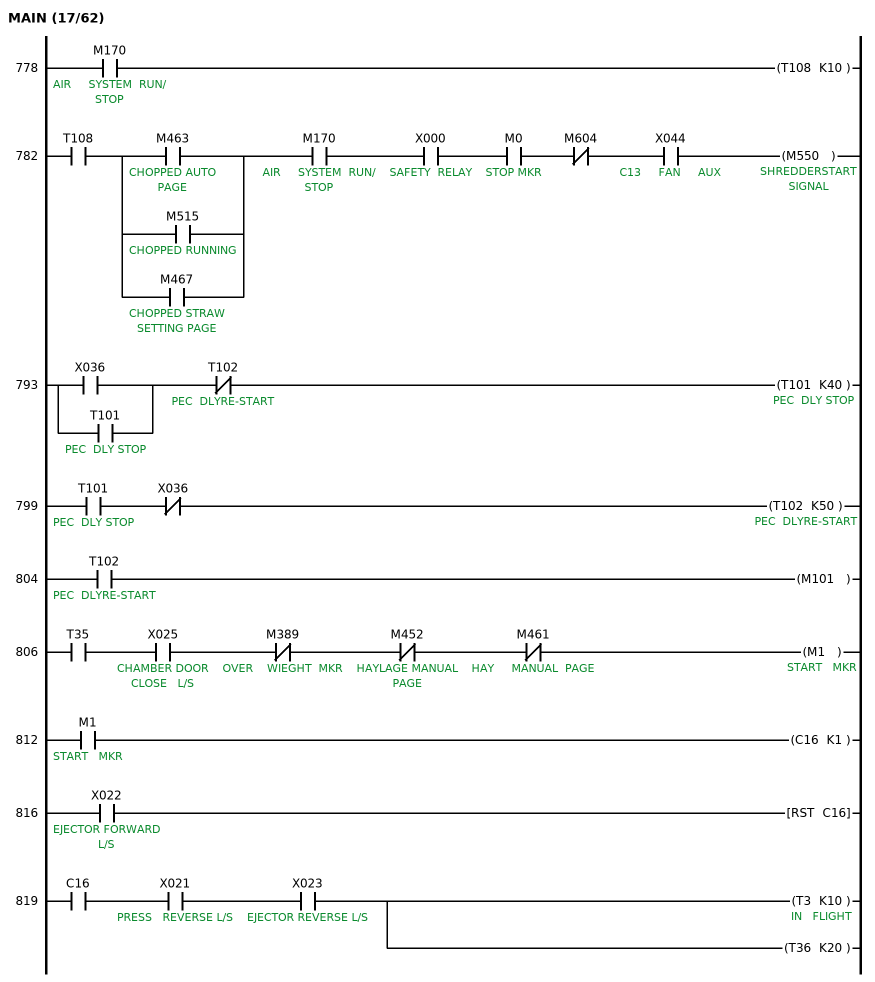
778   LD      M170  ; AIR     SYSTEM  RUN/    STOP
      OUT     T108 K10
782   LD      T108
      LD      M463  ; CHOPPED AUTO    PAGE
      OR      M515  ; CHOPPED RUNNING
      OR      M467  ; CHOPPED STRAW   SETTING PAGE
      ANB
      AND     M170  ; AIR     SYSTEM  RUN/    STOP
      AND     X000  ; SAFETY  RELAY
      AND     M0  ; STOP MKR
      ANI     M604
      AND     X044  ; C13     FAN     AUX
      OUT     M550  ; SHREDDERSTART   SIGNAL
793   LD      X036
      OR      T101  ; PEC  DLY STOP
      ANI     T102  ; PEC  DLYRE-START
      OUT     T101 K40  ; PEC  DLY STOP
799   LD      T101  ; PEC  DLY STOP
      ANI     X036
      OUT     T102 K50  ; PEC  DLYRE-START
804   LD      T102  ; PEC  DLYRE-START
      OUT     M101
806   LD      T35
      AND     X025  ; CHAMBER DOOR    CLOSE   L/S
      ANI     M389  ; OVER    WIEGHT  MKR
      ANI     M452  ; HAYLAGE MANUAL  PAGE
      ANI     M461  ; HAY     MANUAL  PAGE
      OUT     M1  ; START   MKR
812   LD      M1  ; START   MKR
      OUT     C16 K1
816   LD      X022  ; EJECTOR FORWARD L/S
      RST     C16
819   LD      C16
      AND     X021  ; PRESS   REVERSE L/S
      AND     X023  ; EJECTOR REVERSE L/S
      OUT     T3 K10  ; IN   FLIGHT
      OUT     T36 K20
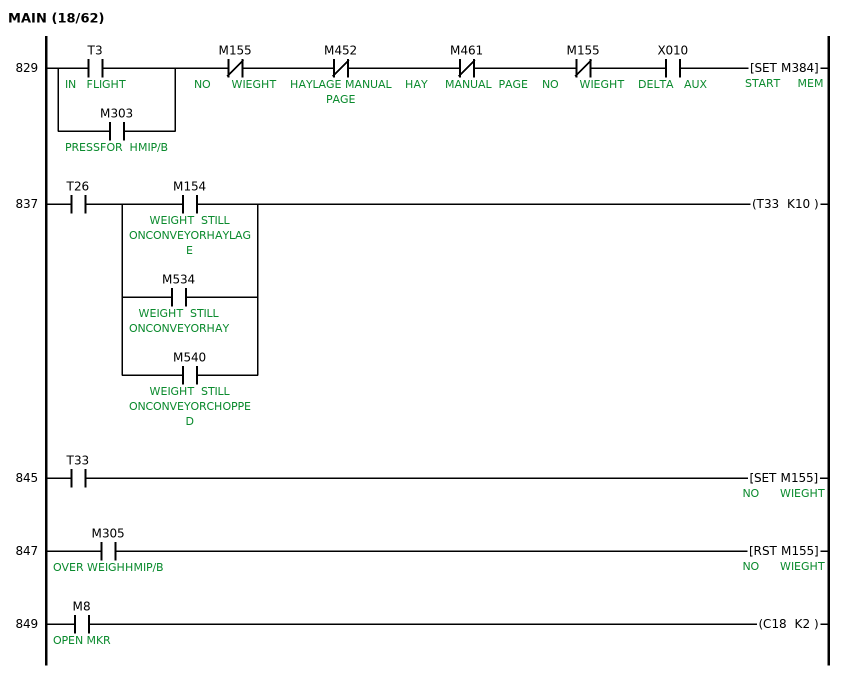
829   LD      T3  ; IN   FLIGHT
      OR      M303  ; PRESSFOR  HMIP/B
      ANI     M155  ; NO      WIEGHT
      ANI     M452  ; HAYLAGE MANUAL  PAGE
      ANI     M461  ; HAY     MANUAL  PAGE
      ANI     M155  ; NO      WIEGHT
      AND     X010  ; DELTA   AUX
      SET     M384  ; START     MEM
837   LD      T26
      LD      M154  ; WEIGHT  STILL ONCONVEYORHAYLAGE
      OR      M534  ; WEIGHT  STILL ONCONVEYORHAY
      OR      M540  ; WEIGHT  STILL ONCONVEYORCHOPPED
      ANB
      OUT     T33 K10
845   LD      T33
      SET     M155  ; NO      WIEGHT
847   LD      M305  ; OVER WEIGHHMIP/B
      RST     M155  ; NO      WIEGHT
849   LD      M8  ; OPEN MKR
      OUT     C18 K2
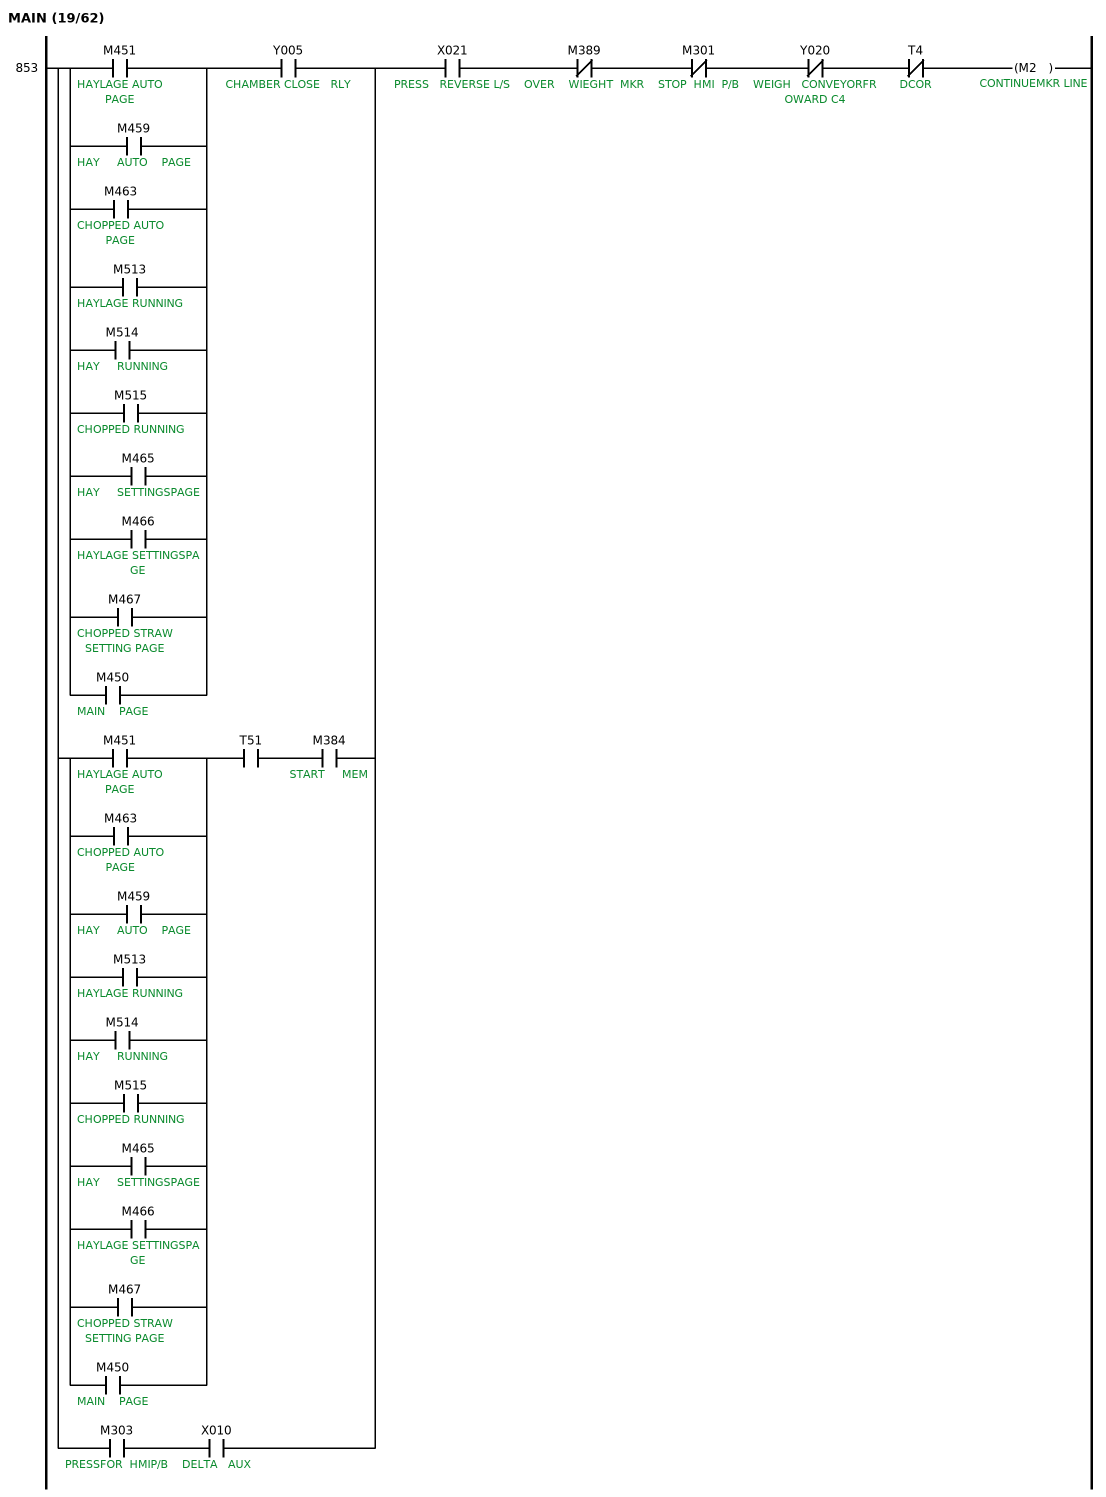
853   LD      M451  ; HAYLAGE AUTO    PAGE
      OR      M459  ; HAY     AUTO    PAGE
      OR      M463  ; CHOPPED AUTO    PAGE
      OR      M513  ; HAYLAGE RUNNING
      OR      M514  ; HAY     RUNNING
      OR      M515  ; CHOPPED RUNNING
      OR      M465  ; HAY     SETTINGSPAGE
      OR      M466  ; HAYLAGE SETTINGSPAGE
      OR      M467  ; CHOPPED STRAW   SETTING PAGE
      OR      M450  ; MAIN    PAGE
      AND     Y005  ; CHAMBER CLOSE   RLY
      LD      M451  ; HAYLAGE AUTO    PAGE
      OR      M463  ; CHOPPED AUTO    PAGE
      OR      M459  ; HAY     AUTO    PAGE
      OR      M513  ; HAYLAGE RUNNING
      OR      M514  ; HAY     RUNNING
      OR      M515  ; CHOPPED RUNNING
      OR      M465  ; HAY     SETTINGSPAGE
      OR      M466  ; HAYLAGE SETTINGSPAGE
      OR      M467  ; CHOPPED STRAW   SETTING PAGE
      OR      M450  ; MAIN    PAGE
      AND     T51
      AND     M384  ; START     MEM
      ORB
      LD      M303  ; PRESSFOR  HMIP/B
      AND     X010  ; DELTA   AUX
      ORB
      AND     X021  ; PRESS   REVERSE L/S
      ANI     M389  ; OVER    WIEGHT  MKR
      ANI     M301  ; STOP  HMI  P/B
      ANI     Y020  ; WEIGH   CONVEYORFROWARD C4
      ANI     T4  ; DCOR
      OUT     M2  ; CONTINUEMKR LINE
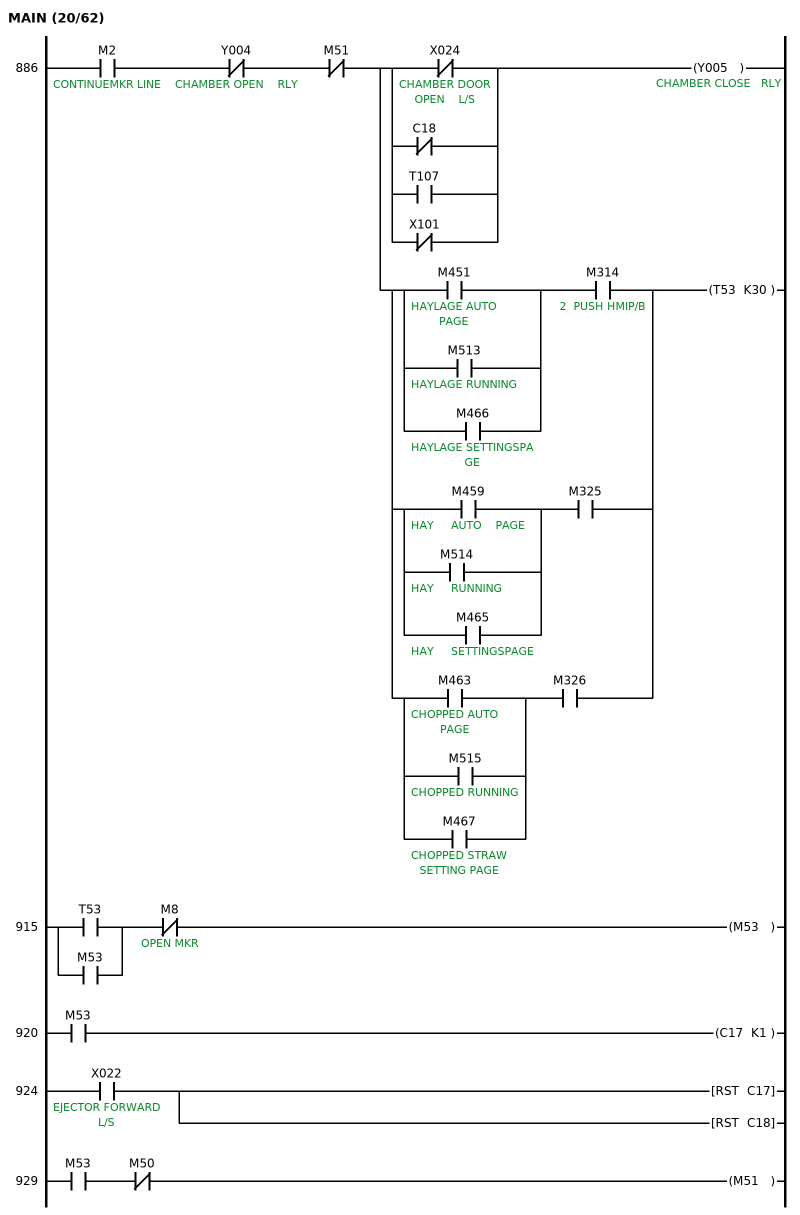
886   LD      M2  ; CONTINUEMKR LINE
      ANI     Y004  ; CHAMBER OPEN    RLY
      ANI     M51
      MPS
      LDI     X024  ; CHAMBER DOOR    OPEN    L/S
      ORI     C18
      OR      T107
      ORI     X101
      ANB
      OUT     Y005  ; CHAMBER CLOSE   RLY
      MPP
      LD      M451  ; HAYLAGE AUTO    PAGE
      OR      M513  ; HAYLAGE RUNNING
      OR      M466  ; HAYLAGE SETTINGSPAGE
      AND     M314  ; 2  PUSH HMIP/B
      LD      M459  ; HAY     AUTO    PAGE
      OR      M514  ; HAY     RUNNING
      OR      M465  ; HAY     SETTINGSPAGE
      AND     M325
      ORB
      LD      M463  ; CHOPPED AUTO    PAGE
      OR      M515  ; CHOPPED RUNNING
      OR      M467  ; CHOPPED STRAW   SETTING PAGE
      AND     M326
      ORB
      ANB
      OUT     T53 K30
915   LD      T53
      OR      M53
      ANI     M8  ; OPEN MKR
      OUT     M53
920   LD      M53
      OUT     C17 K1
924   LD      X022  ; EJECTOR FORWARD L/S
      RST     C17
      RST     C18
929   LD      M53
      ANI     M50
      OUT     M51
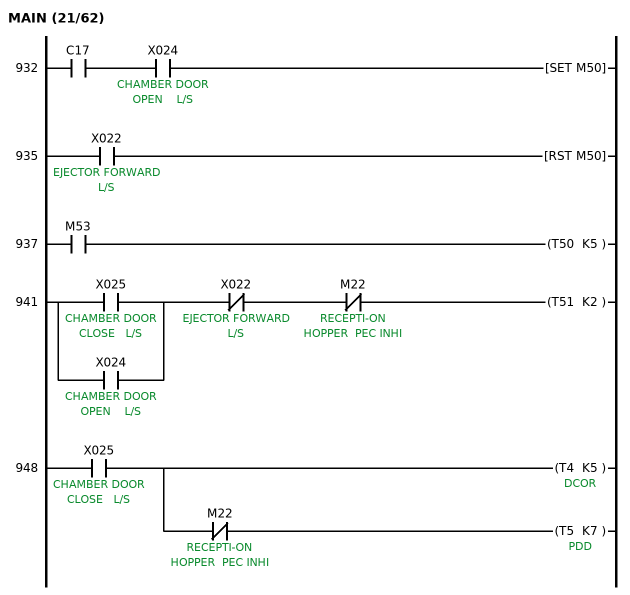
932   LD      C17
      AND     X024  ; CHAMBER DOOR    OPEN    L/S
      SET     M50
935   LD      X022  ; EJECTOR FORWARD L/S
      RST     M50
937   LD      M53
      OUT     T50 K5
941   LD      X025  ; CHAMBER DOOR    CLOSE   L/S
      OR      X024  ; CHAMBER DOOR    OPEN    L/S
      ANI     X022  ; EJECTOR FORWARD L/S
      ANI     M22  ; RECEPTI-ON      HOPPER  PEC INHI
      OUT     T51 K2
948   LD      X025  ; CHAMBER DOOR    CLOSE   L/S
      OUT     T4 K5  ; DCOR
      ANI     M22  ; RECEPTI-ON      HOPPER  PEC INHI
      OUT     T5 K7  ; PDD
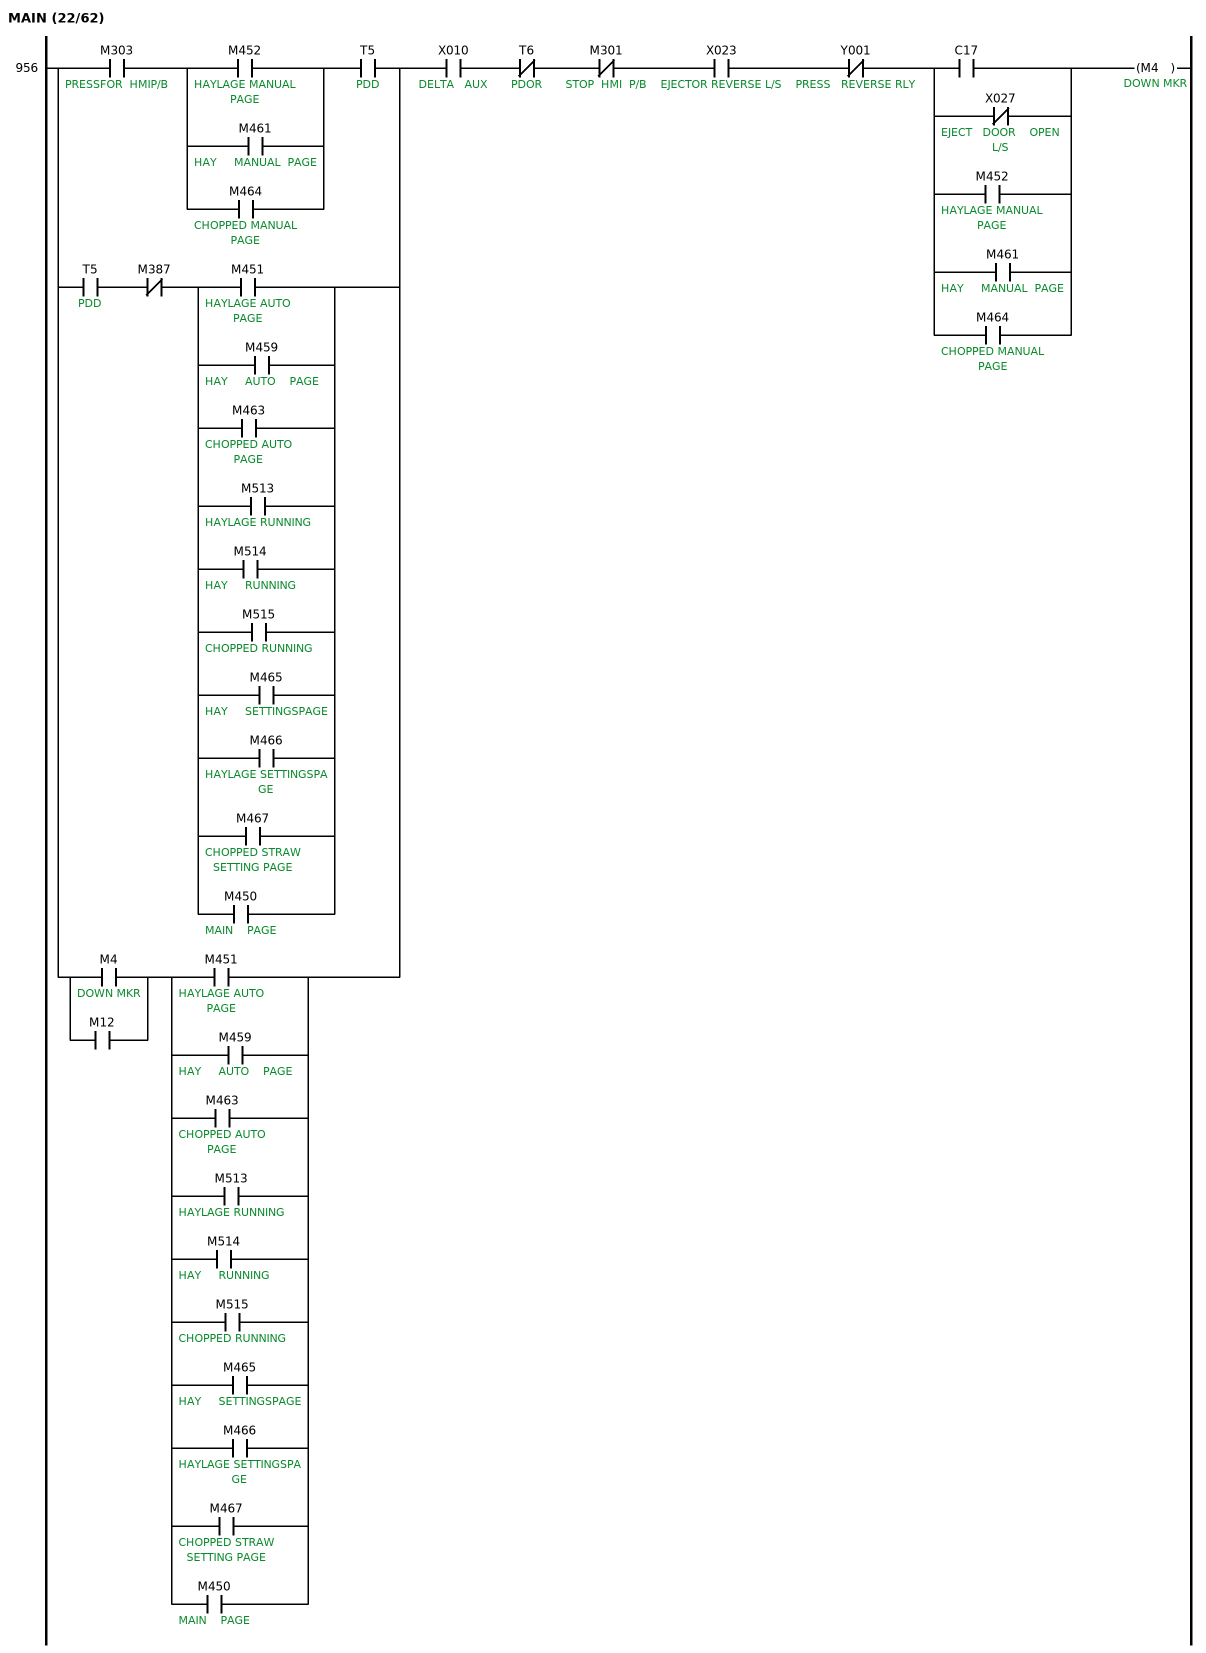
956   LD      M303  ; PRESSFOR  HMIP/B
      LD      M452  ; HAYLAGE MANUAL  PAGE
      OR      M461  ; HAY     MANUAL  PAGE
      OR      M464  ; CHOPPED MANUAL  PAGE
      ANB
      AND     T5  ; PDD
      LD      T5  ; PDD
      ANI     M387
      LD      M451  ; HAYLAGE AUTO    PAGE
      OR      M459  ; HAY     AUTO    PAGE
      OR      M463  ; CHOPPED AUTO    PAGE
      OR      M513  ; HAYLAGE RUNNING
      OR      M514  ; HAY     RUNNING
      OR      M515  ; CHOPPED RUNNING
      OR      M465  ; HAY     SETTINGSPAGE
      OR      M466  ; HAYLAGE SETTINGSPAGE
      OR      M467  ; CHOPPED STRAW   SETTING PAGE
      OR      M450  ; MAIN    PAGE
      ANB
      ORB
      LD      M4  ; DOWN MKR
      OR      M12
      LD      M451  ; HAYLAGE AUTO    PAGE
      OR      M459  ; HAY     AUTO    PAGE
      OR      M463  ; CHOPPED AUTO    PAGE
      OR      M513  ; HAYLAGE RUNNING
      OR      M514  ; HAY     RUNNING
      OR      M515  ; CHOPPED RUNNING
      OR      M465  ; HAY     SETTINGSPAGE
      OR      M466  ; HAYLAGE SETTINGSPAGE
      OR      M467  ; CHOPPED STRAW   SETTING PAGE
      OR      M450  ; MAIN    PAGE
      ANB
      ORB
      AND     X010  ; DELTA   AUX
      ANI     T6  ; PDOR
      ANI     M301  ; STOP  HMI  P/B
      AND     X023  ; EJECTOR REVERSE L/S
      ANI     Y001  ; PRESS   REVERSE RLY
      LD      C17
      ORI     X027  ; EJECT   DOOR    OPEN L/S
      OR      M452  ; HAYLAGE MANUAL  PAGE
      OR      M461  ; HAY     MANUAL  PAGE
      OR      M464  ; CHOPPED MANUAL  PAGE
      ANB
      OUT     M4  ; DOWN MKR
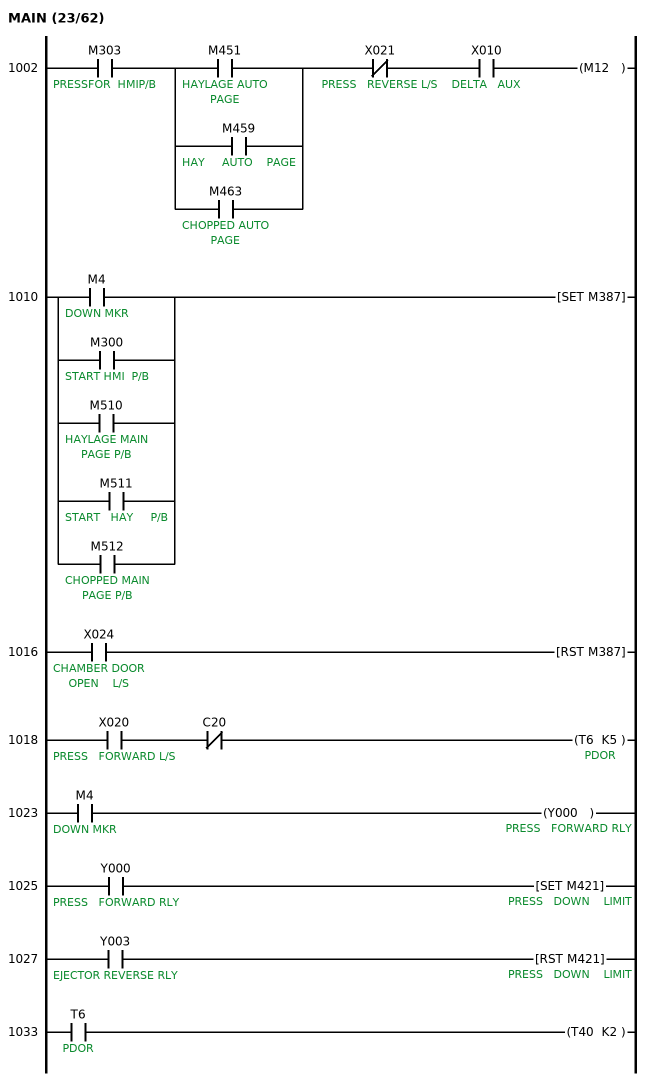
1002  LD      M303  ; PRESSFOR  HMIP/B
      LD      M451  ; HAYLAGE AUTO    PAGE
      OR      M459  ; HAY     AUTO    PAGE
      OR      M463  ; CHOPPED AUTO    PAGE
      ANB
      ANI     X021  ; PRESS   REVERSE L/S
      AND     X010  ; DELTA   AUX
      OUT     M12
1010  LD      M4  ; DOWN MKR
      OR      M300  ; START HMI  P/B
      OR      M510  ; HAYLAGE MAIN    PAGE P/B
      OR      M511  ; START   HAY     P/B
      OR      M512  ; CHOPPED MAIN    PAGE P/B
      SET     M387
1016  LD      X024  ; CHAMBER DOOR    OPEN    L/S
      RST     M387
1018  LD      X020  ; PRESS   FORWARD L/S
      ANI     C20
      OUT     T6 K5  ; PDOR
1023  LD      M4  ; DOWN MKR
      OUT     Y000  ; PRESS   FORWARD RLY
1025  LD      Y000  ; PRESS   FORWARD RLY
      SET     M421  ; PRESS   DOWN    LIMIT
1027  LD      Y003  ; EJECTOR REVERSE RLY
      RST     M421  ; PRESS   DOWN    LIMIT
1033  LD      T6  ; PDOR
      OUT     T40 K2
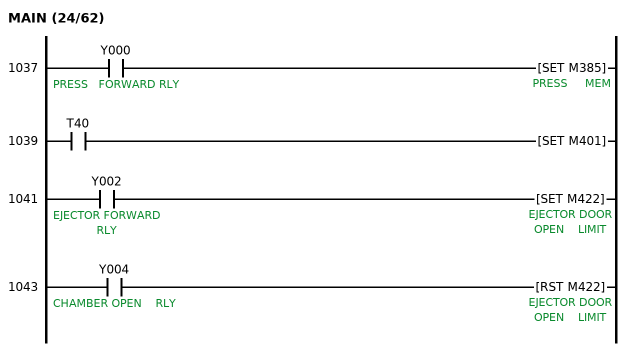
1037  LD      Y000  ; PRESS   FORWARD RLY
      SET     M385  ; PRESS     MEM
1039  LD      T40
      SET     M401
1041  LD      Y002  ; EJECTOR FORWARD RLY
      SET     M422  ; EJECTOR DOOR    OPEN    LIMIT
1043  LD      Y004  ; CHAMBER OPEN    RLY
      RST     M422  ; EJECTOR DOOR    OPEN    LIMIT
